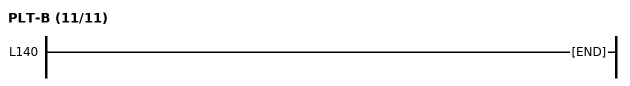
; L140
END

PROGRAM NG_CHUTE (task: 스캔 프로그램)

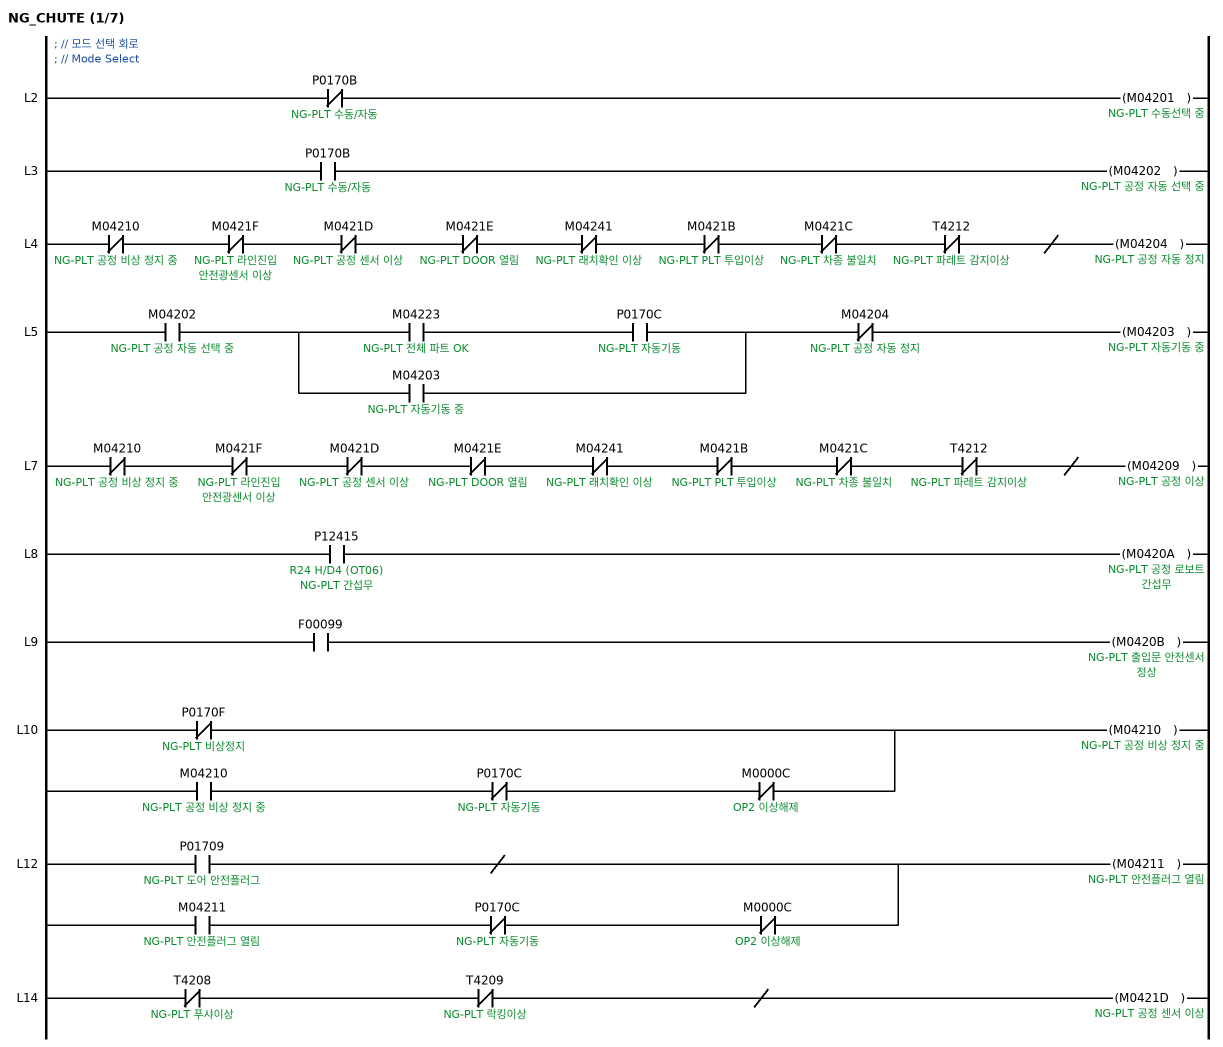
// // 모드 선택 회로
//   // Mode Select
; L2
LOAD NOT  P0170B	// NG-PLT 수동/자동
OUT       M04201	// NG-PLT 수동선택 중
; L3
LOAD      P0170B	// NG-PLT 수동/자동
OUT       M04202	// NG-PLT 공정 자동 선택 중
; L4
LOAD NOT  M04210	// NG-PLT 공정 비상 정지 중
AND NOT   M0421F	// NG-PLT 라인진입 안전광센서 이상
AND NOT   M0421D	// NG-PLT 공정 센서 이상
AND NOT   M0421E	// NG-PLT DOOR 열림
AND NOT   M04241	// NG-PLT 래치확인 이상
AND NOT   M0421B	// NG-PLT PLT 투입이상
AND NOT   M0421C	// NG-PLT 차종 불일치
AND NOT   T4212	// NG-PLT 파레트 감지이상
NOT
OUT       M04204	// NG-PLT 공정 자동 정지
; L5
LOAD      M04202	// NG-PLT 공정 자동 선택 중
LOAD      M04223	// NG-PLT 전체 파트 OK
AND       P0170C	// NG-PLT 자동기동
OR        M04203	// NG-PLT 자동기동 중
AND LOAD
AND NOT   M04204	// NG-PLT 공정 자동 정지
OUT       M04203	// NG-PLT 자동기동 중
; L7
LOAD NOT  M04210	// NG-PLT 공정 비상 정지 중
AND NOT   M0421F	// NG-PLT 라인진입 안전광센서 이상
AND NOT   M0421D	// NG-PLT 공정 센서 이상
AND NOT   M0421E	// NG-PLT DOOR 열림
AND NOT   M04241	// NG-PLT 래치확인 이상
AND NOT   M0421B	// NG-PLT PLT 투입이상
AND NOT   M0421C	// NG-PLT 차종 불일치
AND NOT   T4212	// NG-PLT 파레트 감지이상
NOT
OUT       M04209	// NG-PLT 공정 이상
; L8
LOAD      P12415	// R24 H/D4 (OT06) NG-PLT 간섭무
OUT       M0420A	// NG-PLT 공정 로보트 간섭무
; L9
LOAD      F00099
OUT       M0420B	// NG-PLT 출입문 안전센서 정상
; L10
LOAD NOT  P0170F	// NG-PLT 비상정지
LOAD      M04210	// NG-PLT 공정 비상 정지 중
AND NOT   P0170C	// NG-PLT 자동기동
AND NOT   M0000C	// OP2 이상해제
OR LOAD
OUT       M04210	// NG-PLT 공정 비상 정지 중
; L12
LOAD      P01709	// NG-PLT 도어 안전플러그
NOT
LOAD      M04211	// NG-PLT 안전플러그 열림
AND NOT   P0170C	// NG-PLT 자동기동
AND NOT   M0000C	// OP2 이상해제
OR LOAD
OUT       M04211	// NG-PLT 안전플러그 열림
; L14
LOAD NOT  T4208	// NG-PLT 푸샤이상
AND NOT   T4209	// NG-PLT 락킹이상
NOT
OUT       M0421D	// NG-PLT 공정 센서 이상

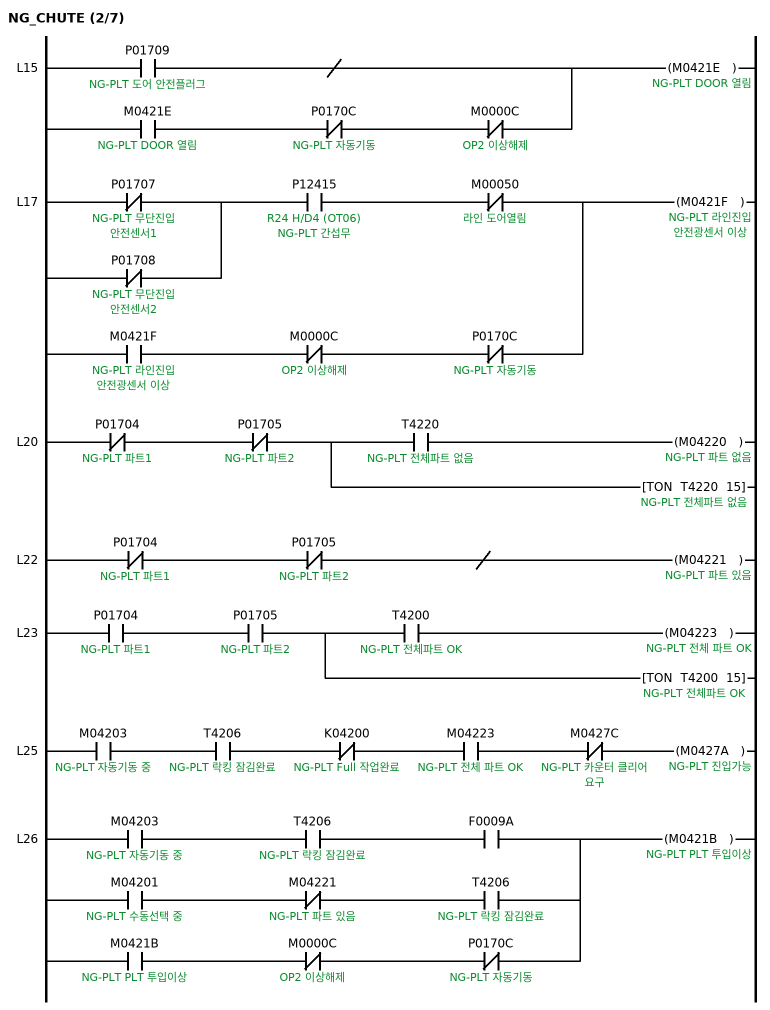
; L15
LOAD      P01709	// NG-PLT 도어 안전플러그
NOT
LOAD      M0421E	// NG-PLT DOOR 열림
AND NOT   P0170C	// NG-PLT 자동기동
AND NOT   M0000C	// OP2 이상해제
OR LOAD
OUT       M0421E	// NG-PLT DOOR 열림
; L17
LOAD NOT  P01707	// NG-PLT 무단진입 안전센서1
OR NOT    P01708	// NG-PLT 무단진입 안전센서2
AND       P12415	// R24 H/D4 (OT06) NG-PLT 간섭무
AND NOT   M00050	// 라인 도어열림
LOAD      M0421F	// NG-PLT 라인진입 안전광센서 이상
AND NOT   M0000C	// OP2 이상해제
AND NOT   P0170C	// NG-PLT 자동기동
OR LOAD
OUT       M0421F	// NG-PLT 라인진입 안전광센서 이상
; L20
LOAD NOT  P01704	// NG-PLT 파트1
AND NOT   P01705	// NG-PLT 파트2
MPUSH
AND       T4220	// NG-PLT 전체파트 없음
OUT       M04220	// NG-PLT 파트 없음
MPOP
TON       T4220 15	// NG-PLT 전체파트 없음
; L22
LOAD NOT  P01704	// NG-PLT 파트1
AND NOT   P01705	// NG-PLT 파트2
NOT
OUT       M04221	// NG-PLT 파트 있음
; L23
LOAD      P01704	// NG-PLT 파트1
AND       P01705	// NG-PLT 파트2
MPUSH
AND       T4200	// NG-PLT 전체파트 OK
OUT       M04223	// NG-PLT 전체 파트 OK
MPOP
TON       T4200 15	// NG-PLT 전체파트 OK
; L25
LOAD      M04203	// NG-PLT 자동기동 중
AND       T4206	// NG-PLT 락킹 잠김완료
AND NOT   K04200	// NG-PLT Full 작업완료
AND       M04223	// NG-PLT 전체 파트 OK
AND NOT   M0427C	// NG-PLT 카운터 클리어 요구
OUT       M0427A	// NG-PLT 진입가능
; L26
LOAD      M04203	// NG-PLT 자동기동 중
AND       T4206	// NG-PLT 락킹 잠김완료
AND       F0009A
LOAD      M04201	// NG-PLT 수동선택 중
AND NOT   M04221	// NG-PLT 파트 있음
AND       T4206	// NG-PLT 락킹 잠김완료
OR LOAD
LOAD      M0421B	// NG-PLT PLT 투입이상
AND NOT   M0000C	// OP2 이상해제
AND NOT   P0170C	// NG-PLT 자동기동
OR LOAD
OUT       M0421B	// NG-PLT PLT 투입이상

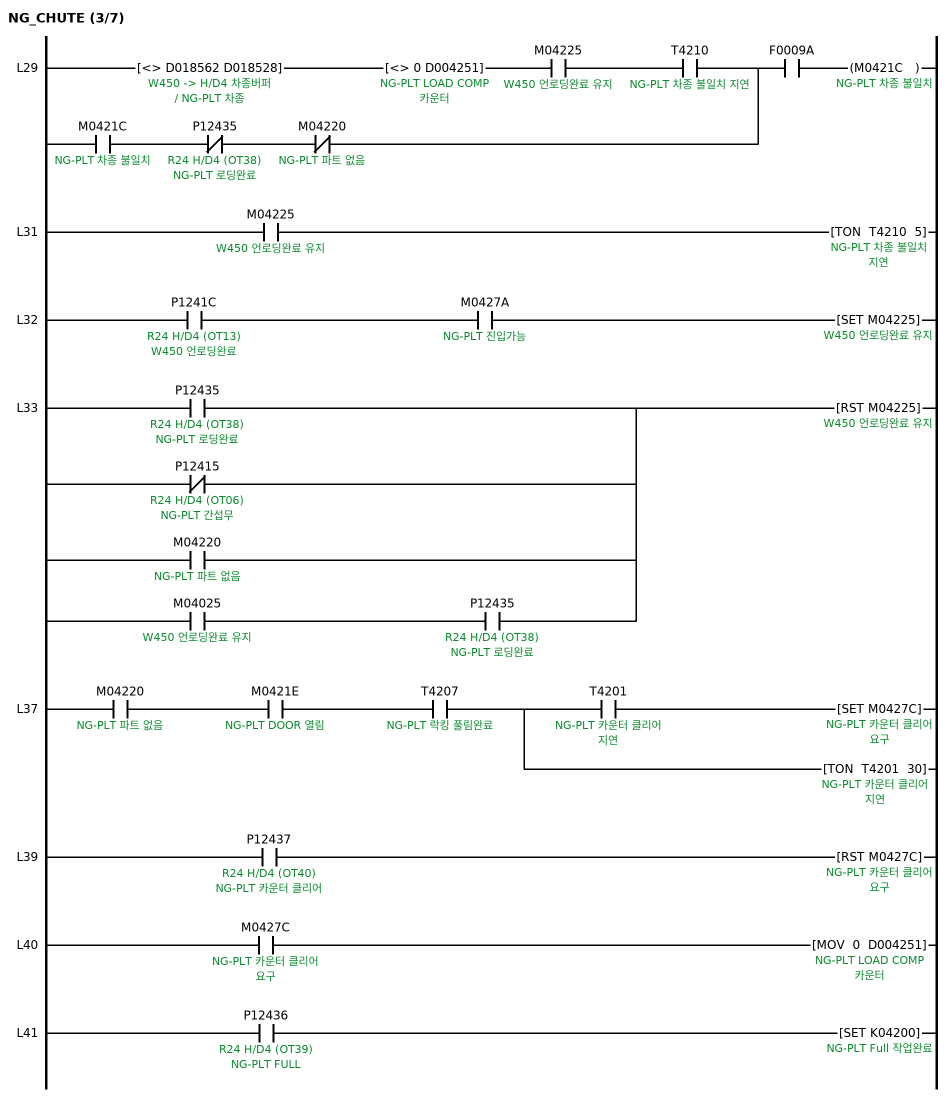
; L29
LOAD<>    D018562 D018528	// W450 -> H/D4 차종버퍼 / NG-PLT 차종
AND<>     0 D004251	// NG-PLT LOAD COMP 카운터
AND       M04225	// W450 언로딩완료 유지
AND       T4210	// NG-PLT 차종 불일치 지연
LOAD      M0421C	// NG-PLT 차종 불일치
AND NOT   P12435	// R24 H/D4 (OT38) NG-PLT 로딩완료
AND NOT   M04220	// NG-PLT 파트 없음
OR LOAD
AND       F0009A
OUT       M0421C	// NG-PLT 차종 불일치
; L31
LOAD      M04225	// W450 언로딩완료 유지
TON       T4210 5	// NG-PLT 차종 불일치 지연
; L32
LOAD      P1241C	// R24 H/D4 (OT13) W450 언로딩완료
AND       M0427A	// NG-PLT 진입가능
SET       M04225	// W450 언로딩완료 유지
; L33
LOAD      P12435	// R24 H/D4 (OT38) NG-PLT 로딩완료
OR NOT    P12415	// R24 H/D4 (OT06) NG-PLT 간섭무
OR        M04220	// NG-PLT 파트 없음
LOAD      M04025	// W450 언로딩완료 유지
AND       P12435	// R24 H/D4 (OT38) NG-PLT 로딩완료
OR LOAD
RST       M04225	// W450 언로딩완료 유지
; L37
LOAD      M04220	// NG-PLT 파트 없음
AND       M0421E	// NG-PLT DOOR 열림
AND       T4207	// NG-PLT 락킹 풀림완료
MPUSH
AND       T4201	// NG-PLT 카운터 클리어 지연
SET       M0427C	// NG-PLT 카운터 클리어 요구
MPOP
TON       T4201 30	// NG-PLT 카운터 클리어 지연
; L39
LOAD      P12437	// R24 H/D4 (OT40) NG-PLT 카운터 클리어
RST       M0427C	// NG-PLT 카운터 클리어 요구
; L40
LOAD      M0427C	// NG-PLT 카운터 클리어 요구
MOV       0 D004251	// NG-PLT LOAD COMP 카운터
; L41
LOAD      P12436	// R24 H/D4 (OT39) NG-PLT FULL
SET       K04200	// NG-PLT Full 작업완료

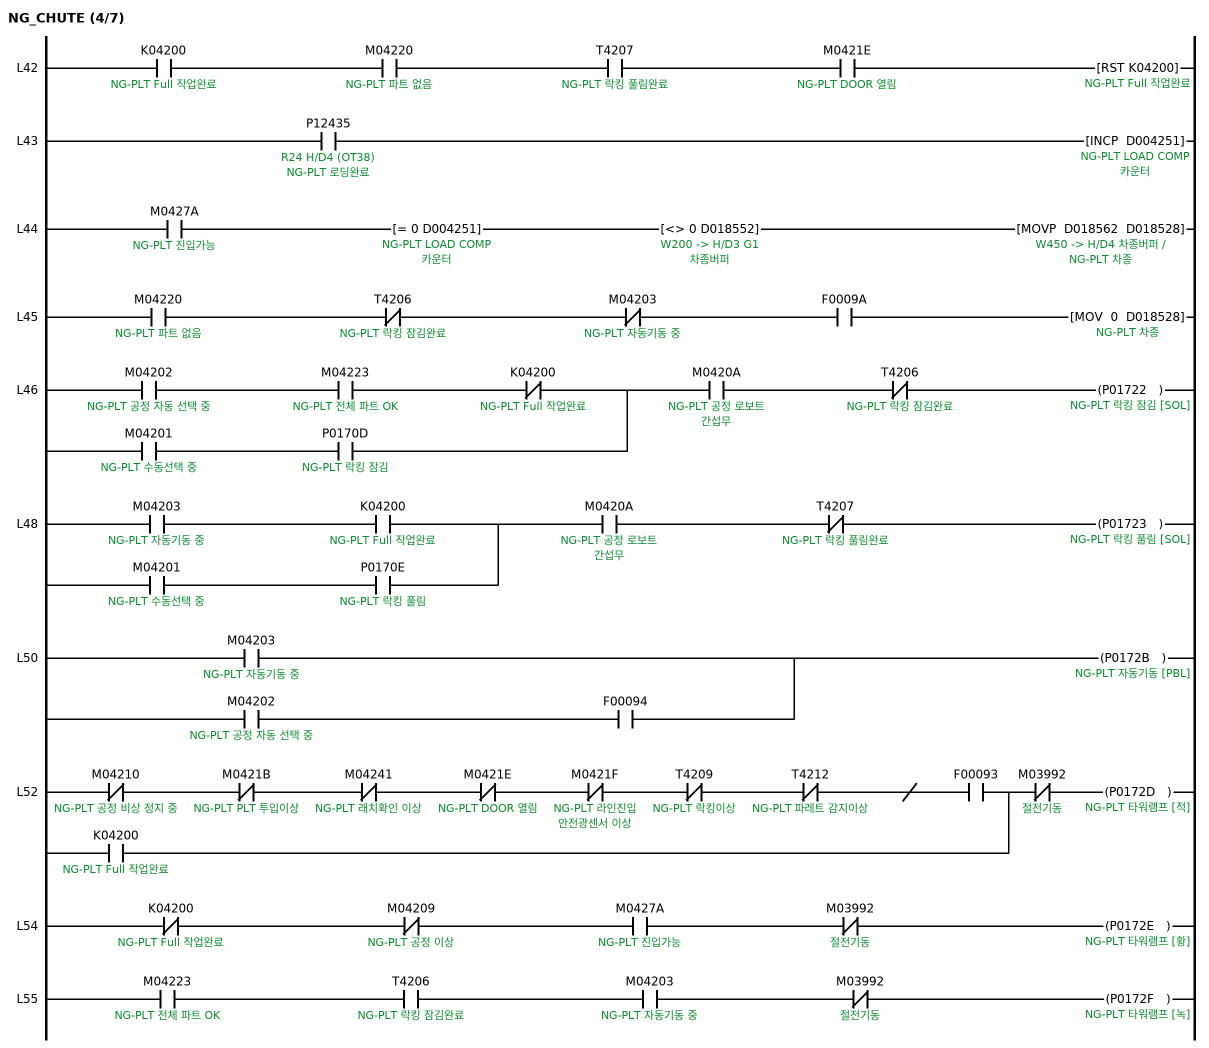
; L42
LOAD      K04200	// NG-PLT Full 작업완료
AND       M04220	// NG-PLT 파트 없음
AND       T4207	// NG-PLT 락킹 풀림완료
AND       M0421E	// NG-PLT DOOR 열림
RST       K04200	// NG-PLT Full 작업완료
; L43
LOAD      P12435	// R24 H/D4 (OT38) NG-PLT 로딩완료
INCP      D004251	// NG-PLT LOAD COMP 카운터
; L44
LOAD      M0427A	// NG-PLT 진입가능
AND=      0 D004251	// NG-PLT LOAD COMP 카운터
AND<>     0 D018552	// W200 -> H/D3 G1 차종버퍼
MOVP      D018562 D018528	// W450 -> H/D4 차종버퍼 / NG-PLT 차종
; L45
LOAD      M04220	// NG-PLT 파트 없음
AND NOT   T4206	// NG-PLT 락킹 잠김완료
AND NOT   M04203	// NG-PLT 자동기동 중
AND       F0009A
MOV       0 D018528	// NG-PLT 차종
; L46
LOAD      M04202	// NG-PLT 공정 자동 선택 중
AND       M04223	// NG-PLT 전체 파트 OK
AND NOT   K04200	// NG-PLT Full 작업완료
LOAD      M04201	// NG-PLT 수동선택 중
AND       P0170D	// NG-PLT 락킹 잠김
OR LOAD
AND       M0420A	// NG-PLT 공정 로보트 간섭무
AND NOT   T4206	// NG-PLT 락킹 잠김완료
OUT       P01722	// NG-PLT 락킹 잠김 [SOL]
; L48
LOAD      M04203	// NG-PLT 자동기동 중
AND       K04200	// NG-PLT Full 작업완료
LOAD      M04201	// NG-PLT 수동선택 중
AND       P0170E	// NG-PLT 락킹 풀림
OR LOAD
AND       M0420A	// NG-PLT 공정 로보트 간섭무
AND NOT   T4207	// NG-PLT 락킹 풀림완료
OUT       P01723	// NG-PLT 락킹 풀림 [SOL]
; L50
LOAD      M04203	// NG-PLT 자동기동 중
LOAD      M04202	// NG-PLT 공정 자동 선택 중
AND       F00094
OR LOAD
OUT       P0172B	// NG-PLT 자동기동 [PBL]
; L52
LOAD NOT  M04210	// NG-PLT 공정 비상 정지 중
AND NOT   M0421B	// NG-PLT PLT 투입이상
AND NOT   M04241	// NG-PLT 래치확인 이상
AND NOT   M0421E	// NG-PLT DOOR 열림
AND NOT   M0421F	// NG-PLT 라인진입 안전광센서 이상
AND NOT   T4209	// NG-PLT 락킹이상
AND NOT   T4212	// NG-PLT 파레트 감지이상
NOT
AND       F00093
OR        K04200	// NG-PLT Full 작업완료
AND NOT   M03992	// 절전기동
OUT       P0172D	// NG-PLT 타워램프 [적]
; L54
LOAD NOT  K04200	// NG-PLT Full 작업완료
AND NOT   M04209	// NG-PLT 공정 이상
AND       M0427A	// NG-PLT 진입가능
AND NOT   M03992	// 절전기동
OUT       P0172E	// NG-PLT 타워램프 [황]
; L55
LOAD      M04223	// NG-PLT 전체 파트 OK
AND       T4206	// NG-PLT 락킹 잠김완료
AND       M04203	// NG-PLT 자동기동 중
AND NOT   M03992	// 절전기동
OUT       P0172F	// NG-PLT 타워램프 [녹]

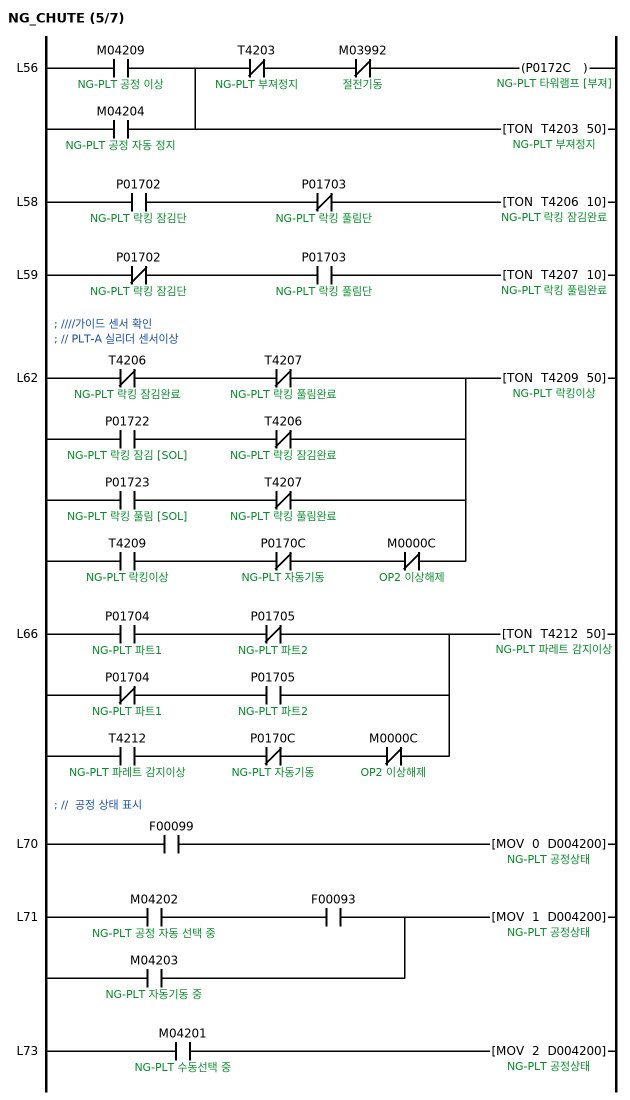
; L56
LOAD      M04209	// NG-PLT 공정 이상
OR        M04204	// NG-PLT 공정 자동 정지
MPUSH
AND NOT   T4203	// NG-PLT 부져정지
AND NOT   M03992	// 절전기동
OUT       P0172C	// NG-PLT 타워램프 [부져]
MPOP
TON       T4203 50	// NG-PLT 부져정지
; L58
LOAD      P01702	// NG-PLT 락킹 잠김단
AND NOT   P01703	// NG-PLT 락킹 풀림단
TON       T4206 10	// NG-PLT 락킹 잠김완료
; L59
LOAD NOT  P01702	// NG-PLT 락킹 잠김단
AND       P01703	// NG-PLT 락킹 풀림단
TON       T4207 10	// NG-PLT 락킹 풀림완료
// ////가이드 센서 확인
// // PLT-A 실리더 센서이상
; L62
LOAD NOT  T4206	// NG-PLT 락킹 잠김완료
AND NOT   T4207	// NG-PLT 락킹 풀림완료
LOAD      P01722	// NG-PLT 락킹 잠김 [SOL]
AND NOT   T4206	// NG-PLT 락킹 잠김완료
OR LOAD
LOAD      P01723	// NG-PLT 락킹 풀림 [SOL]
AND NOT   T4207	// NG-PLT 락킹 풀림완료
OR LOAD
LOAD      T4209	// NG-PLT 락킹이상
AND NOT   P0170C	// NG-PLT 자동기동
AND NOT   M0000C	// OP2 이상해제
OR LOAD
TON       T4209 50	// NG-PLT 락킹이상
; L66
LOAD      P01704	// NG-PLT 파트1
AND NOT   P01705	// NG-PLT 파트2
LOAD NOT  P01704	// NG-PLT 파트1
AND       P01705	// NG-PLT 파트2
OR LOAD
LOAD      T4212	// NG-PLT 파레트 감지이상
AND NOT   P0170C	// NG-PLT 자동기동
AND NOT   M0000C	// OP2 이상해제
OR LOAD
TON       T4212 50	// NG-PLT 파레트 감지이상
//   //  공정 상태 표시
; L70
LOAD      F00099
MOV       0 D004200	// NG-PLT 공정상태
; L71
LOAD      M04202	// NG-PLT 공정 자동 선택 중
AND       F00093
OR        M04203	// NG-PLT 자동기동 중
MOV       1 D004200	// NG-PLT 공정상태
; L73
LOAD      M04201	// NG-PLT 수동선택 중
MOV       2 D004200	// NG-PLT 공정상태

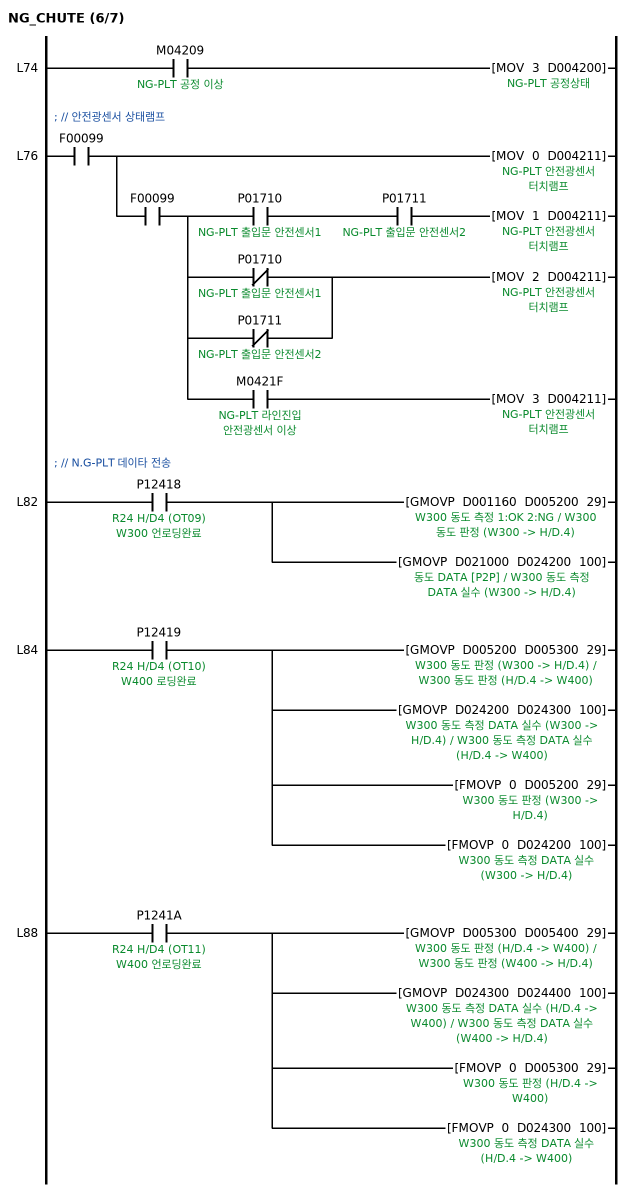
; L74
LOAD      M04209	// NG-PLT 공정 이상
MOV       3 D004200	// NG-PLT 공정상태
//   // 안전광센서 상태램프
; L76
LOAD      F00099
MOV       0 D004211	// NG-PLT 안전광센서 터치램프
AND       F00099
MPUSH
AND       P01710	// NG-PLT 출입문 안전센서1
AND       P01711	// NG-PLT 출입문 안전센서2
MOV       1 D004211	// NG-PLT 안전광센서 터치램프
MLOAD
LOAD NOT  P01710	// NG-PLT 출입문 안전센서1
OR NOT    P01711	// NG-PLT 출입문 안전센서2
AND LOAD
MOV       2 D004211	// NG-PLT 안전광센서 터치램프
MPOP
AND       M0421F	// NG-PLT 라인진입 안전광센서 이상
MOV       3 D004211	// NG-PLT 안전광센서 터치램프
//   // N.G-PLT 데이타 전송
; L82
LOAD      P12418	// R24 H/D4 (OT09) W300 언로딩완료
GMOVP     D001160 D005200 29	// W300 동도 측정 1:OK 2:NG / W300 동도 판정 (W300 -> H/D.4)
GMOVP     D021000 D024200 100	// 동도 DATA [P2P] / W300 동도 측정 DATA 실수 (W300 -> H/D.4)
; L84
LOAD      P12419	// R24 H/D4 (OT10) W400 로딩완료
GMOVP     D005200 D005300 29	// W300 동도 판정 (W300 -> H/D.4) / W300 동도 판정 (H/D.4 -> W400)
GMOVP     D024200 D024300 100	// W300 동도 측정 DATA 실수 (W300 -> H/D.4) / W300 동도 측정 DATA 실수 (H/D.4 -> W400)
FMOVP     0 D005200 29	// W300 동도 판정 (W300 -> H/D.4)
FMOVP     0 D024200 100	// W300 동도 측정 DATA 실수 (W300 -> H/D.4)
; L88
LOAD      P1241A	// R24 H/D4 (OT11) W400 언로딩완료
GMOVP     D005300 D005400 29	// W300 동도 판정 (H/D.4 -> W400) / W300 동도 판정 (W400 -> H/D.4)
GMOVP     D024300 D024400 100	// W300 동도 측정 DATA 실수 (H/D.4 -> W400) / W300 동도 측정 DATA 실수 (W400 -> H/D.4)
FMOVP     0 D005300 29	// W300 동도 판정 (H/D.4 -> W400)
FMOVP     0 D024300 100	// W300 동도 측정 DATA 실수 (H/D.4 -> W400)

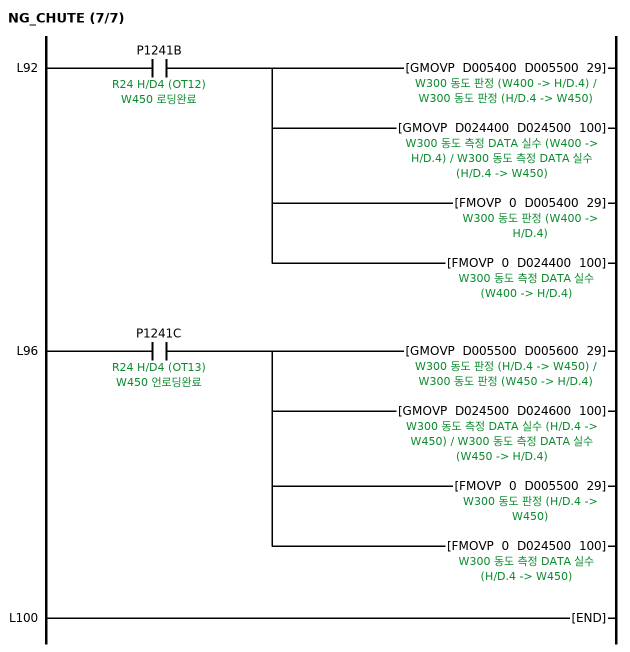
; L92
LOAD      P1241B	// R24 H/D4 (OT12) W450 로딩완료
GMOVP     D005400 D005500 29	// W300 동도 판정 (W400 -> H/D.4) / W300 동도 판정 (H/D.4 -> W450)
GMOVP     D024400 D024500 100	// W300 동도 측정 DATA 실수 (W400 -> H/D.4) / W300 동도 측정 DATA 실수 (H/D.4 -> W450)
FMOVP     0 D005400 29	// W300 동도 판정 (W400 -> H/D.4)
FMOVP     0 D024400 100	// W300 동도 측정 DATA 실수 (W400 -> H/D.4)
; L96
LOAD      P1241C	// R24 H/D4 (OT13) W450 언로딩완료
GMOVP     D005500 D005600 29	// W300 동도 판정 (H/D.4 -> W450) / W300 동도 판정 (W450 -> H/D.4)
GMOVP     D024500 D024600 100	// W300 동도 측정 DATA 실수 (H/D.4 -> W450) / W300 동도 측정 DATA 실수 (W450 -> H/D.4)
FMOVP     0 D005500 29	// W300 동도 판정 (H/D.4 -> W450)
FMOVP     0 D024500 100	// W300 동도 측정 DATA 실수 (H/D.4 -> W450)
; L100
END

PROGRAM OK_NG_Master (task: 스캔 프로그램)

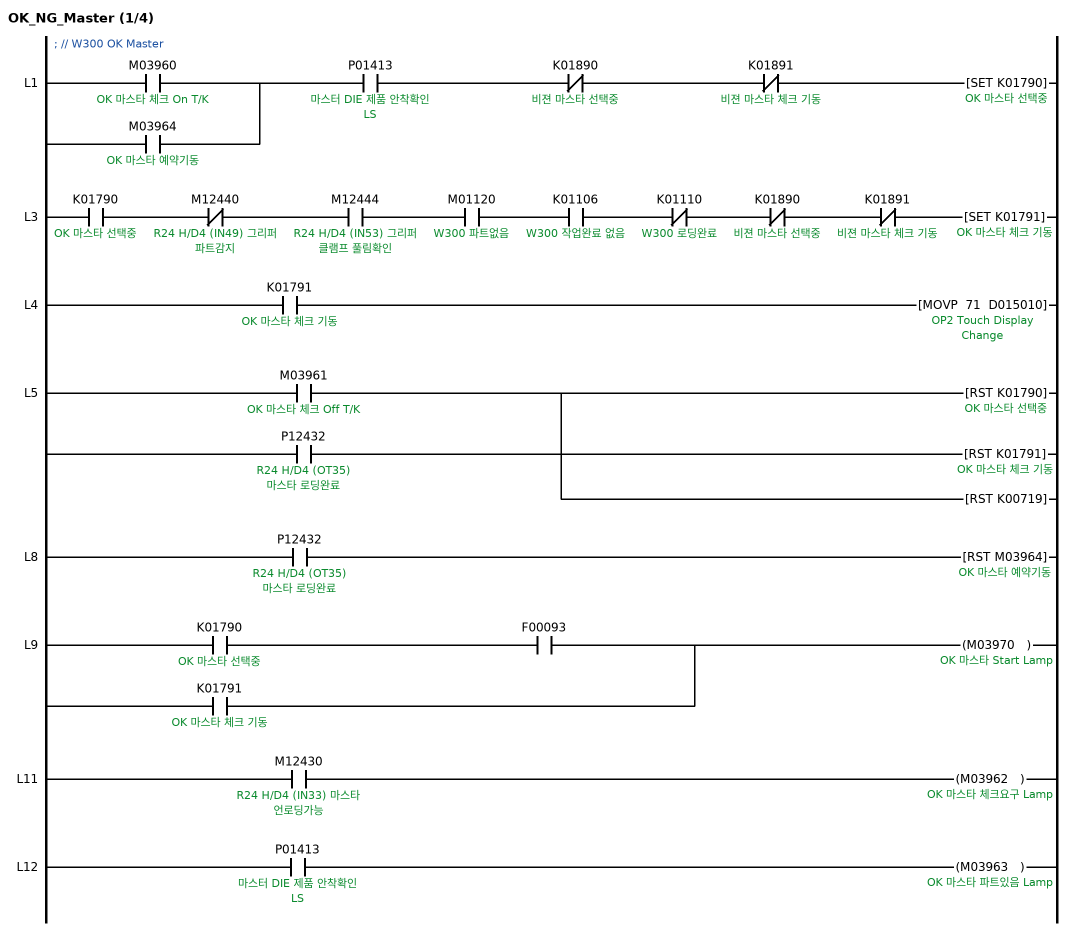
//   // W300 OK Master
; L1
LOAD      M03960	// OK 마스타 체크 On T/K
OR        M03964	// OK 마스타 예약기동
AND       P01413	// 마스터 DIE 제품 안착확인 LS
AND NOT   K01890	// 비젼 마스타 선택중
AND NOT   K01891	// 비젼 마스타 체크 기동
SET       K01790	// OK 마스타 선택중
; L3
LOAD      K01790	// OK 마스타 선택중
AND NOT   M12440	// R24 H/D4 (IN49) 그리퍼 파트감지
AND       M12444	// R24 H/D4 (IN53) 그리퍼 클램프 풀림확인
AND       M01120	// W300 파트없음
AND       K01106	// W300 작업완료 없음
AND NOT   K01110	// W300 로딩완료
AND NOT   K01890	// 비젼 마스타 선택중
AND NOT   K01891	// 비젼 마스타 체크 기동
SET       K01791	// OK 마스타 체크 기동
; L4
LOAD      K01791	// OK 마스타 체크 기동
MOVP      71 D015010	// OP2 Touch Display Change
; L5
LOAD      M03961	// OK 마스타 체크 Off T/K
OR        P12432	// R24 H/D4 (OT35) 마스타 로딩완료
RST       K01790	// OK 마스타 선택중
RST       K01791	// OK 마스타 체크 기동
RST       K00719
; L8
LOAD      P12432	// R24 H/D4 (OT35) 마스타 로딩완료
RST       M03964	// OK 마스타 예약기동
; L9
LOAD      K01790	// OK 마스타 선택중
AND       F00093
OR        K01791	// OK 마스타 체크 기동
OUT       M03970	// OK 마스타 Start Lamp
; L11
LOAD      M12430	// R24 H/D4 (IN33) 마스타 언로딩가능
OUT       M03962	// OK 마스타 체크요구 Lamp
; L12
LOAD      P01413	// 마스터 DIE 제품 안착확인 LS
OUT       M03963	// OK 마스타 파트있음 Lamp

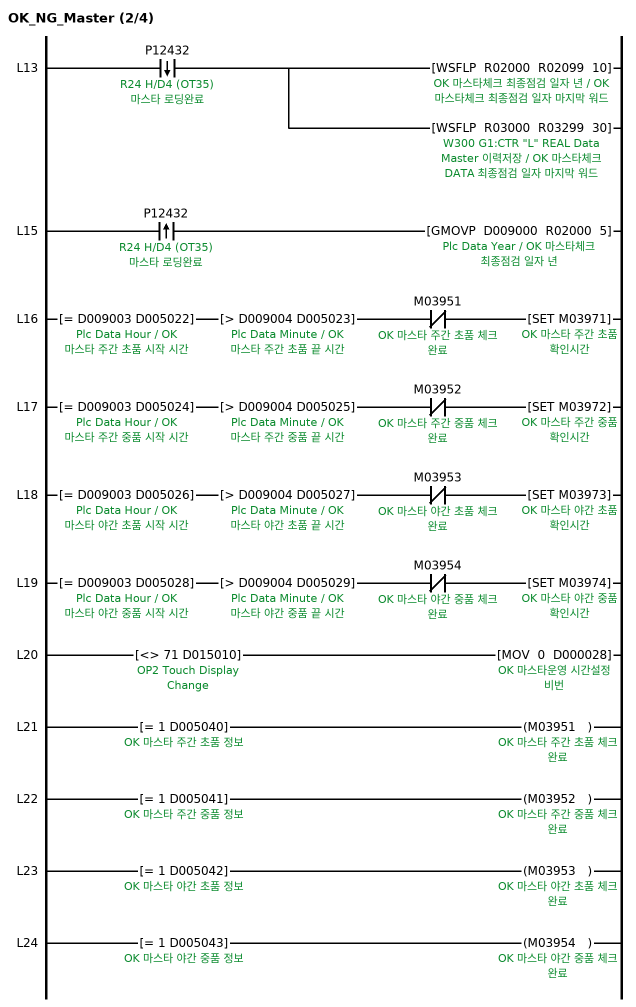
; L13
LOADN     P12432	// R24 H/D4 (OT35) 마스타 로딩완료
WSFLP     R02000 R02099 10	// OK 마스타체크 최종점검 일자 년 / OK 마스타체크 최종점검 일자 마지막 워드
WSFLP     R03000 R03299 30	// W300 G1:CTR "L" REAL Data Master 이력저장 / OK 마스타체크 DATA 최종점검 일자 마지막 워드
; L15
LOADP     P12432	// R24 H/D4 (OT35) 마스타 로딩완료
GMOVP     D009000 R02000 5	// Plc Data Year / OK 마스타체크 최종점검 일자 년
; L16
LOAD=     D009003 D005022	// Plc Data Hour / OK 마스타 주간 초품 시작 시간
AND>      D009004 D005023	// Plc Data Minute / OK 마스타 주간 초품 끝 시간
AND NOT   M03951	// OK 마스타 주간 초품 체크 완료
SET       M03971	// OK 마스타 주간 초품 확인시간
; L17
LOAD=     D009003 D005024	// Plc Data Hour / OK 마스타 주간 중품 시작 시간
AND>      D009004 D005025	// Plc Data Minute / OK 마스타 주간 중품 끝 시간
AND NOT   M03952	// OK 마스타 주간 중품 체크 완료
SET       M03972	// OK 마스타 주간 중품 확인시간
; L18
LOAD=     D009003 D005026	// Plc Data Hour / OK 마스타 야간 초품 시작 시간
AND>      D009004 D005027	// Plc Data Minute / OK 마스타 야간 초품 끝 시간
AND NOT   M03953	// OK 마스타 야간 초품 체크 완료
SET       M03973	// OK 마스타 야간 초품 확인시간
; L19
LOAD=     D009003 D005028	// Plc Data Hour / OK 마스타 야간 중품 시작 시간
AND>      D009004 D005029	// Plc Data Minute / OK 마스타 야간 중품 끝 시간
AND NOT   M03954	// OK 마스타 야간 중품 체크 완료
SET       M03974	// OK 마스타 야간 중품 확인시간
; L20
LOAD<>    71 D015010	// OP2 Touch Display Change
MOV       0 D000028	// OK 마스타운영 시간설정 비번
; L21
LOAD=     1 D005040	// OK 마스타 주간 초품 정보
OUT       M03951	// OK 마스타 주간 초품 체크 완료
; L22
LOAD=     1 D005041	// OK 마스타 주간 중품 정보
OUT       M03952	// OK 마스타 주간 중품 체크 완료
; L23
LOAD=     1 D005042	// OK 마스타 야간 초품 정보
OUT       M03953	// OK 마스타 야간 초품 체크 완료
; L24
LOAD=     1 D005043	// OK 마스타 야간 중품 정보
OUT       M03954	// OK 마스타 야간 중품 체크 완료

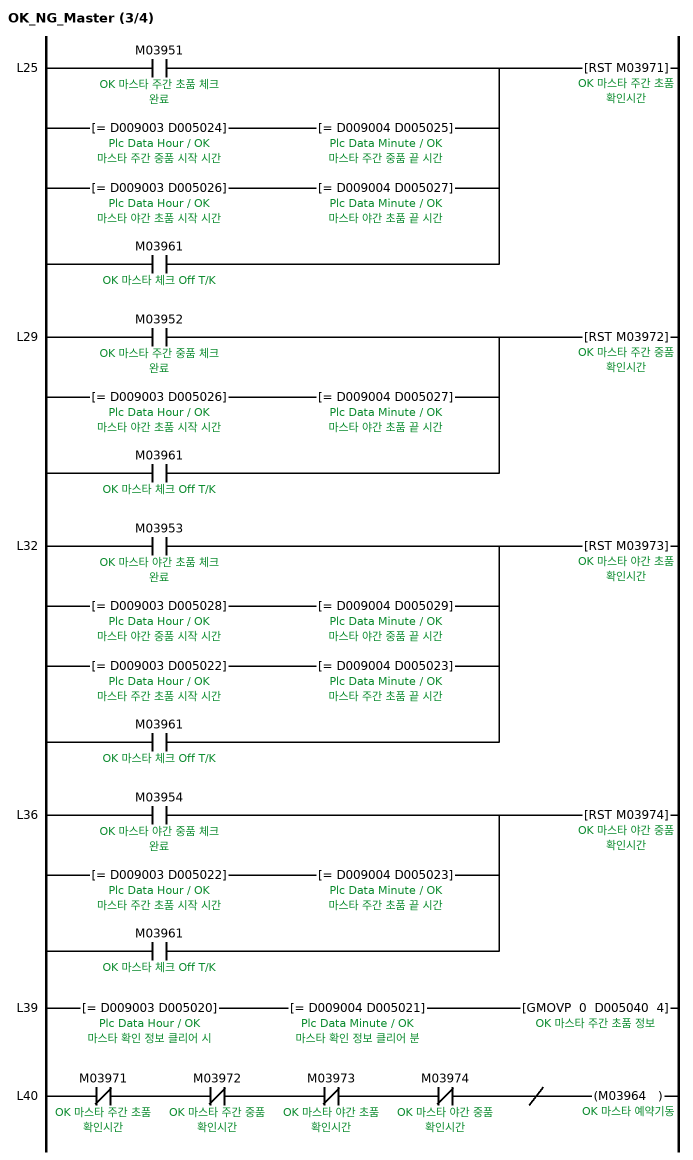
; L25
LOAD      M03951	// OK 마스타 주간 초품 체크 완료
LOAD=     D009003 D005024	// Plc Data Hour / OK 마스타 주간 중품 시작 시간
AND=      D009004 D005025	// Plc Data Minute / OK 마스타 주간 중품 끝 시간
OR LOAD
LOAD=     D009003 D005026	// Plc Data Hour / OK 마스타 야간 초품 시작 시간
AND=      D009004 D005027	// Plc Data Minute / OK 마스타 야간 초품 끝 시간
OR LOAD
OR        M03961	// OK 마스타 체크 Off T/K
RST       M03971	// OK 마스타 주간 초품 확인시간
; L29
LOAD      M03952	// OK 마스타 주간 중품 체크 완료
LOAD=     D009003 D005026	// Plc Data Hour / OK 마스타 야간 초품 시작 시간
AND=      D009004 D005027	// Plc Data Minute / OK 마스타 야간 초품 끝 시간
OR LOAD
OR        M03961	// OK 마스타 체크 Off T/K
RST       M03972	// OK 마스타 주간 중품 확인시간
; L32
LOAD      M03953	// OK 마스타 야간 초품 체크 완료
LOAD=     D009003 D005028	// Plc Data Hour / OK 마스타 야간 중품 시작 시간
AND=      D009004 D005029	// Plc Data Minute / OK 마스타 야간 중품 끝 시간
OR LOAD
LOAD=     D009003 D005022	// Plc Data Hour / OK 마스타 주간 초품 시작 시간
AND=      D009004 D005023	// Plc Data Minute / OK 마스타 주간 초품 끝 시간
OR LOAD
OR        M03961	// OK 마스타 체크 Off T/K
RST       M03973	// OK 마스타 야간 초품 확인시간
; L36
LOAD      M03954	// OK 마스타 야간 중품 체크 완료
LOAD=     D009003 D005022	// Plc Data Hour / OK 마스타 주간 초품 시작 시간
AND=      D009004 D005023	// Plc Data Minute / OK 마스타 주간 초품 끝 시간
OR LOAD
OR        M03961	// OK 마스타 체크 Off T/K
RST       M03974	// OK 마스타 야간 중품 확인시간
; L39
LOAD=     D009003 D005020	// Plc Data Hour / OK 마스타 확인 정보 클리어 시
AND=      D009004 D005021	// Plc Data Minute / OK 마스타 확인 정보 클리어 분
GMOVP     0 D005040 4	// OK 마스타 주간 초품 정보
; L40
LOAD NOT  M03971	// OK 마스타 주간 초품 확인시간
AND NOT   M03972	// OK 마스타 주간 중품 확인시간
AND NOT   M03973	// OK 마스타 야간 초품 확인시간
AND NOT   M03974	// OK 마스타 야간 중품 확인시간
NOT
OUT       M03964	// OK 마스타 예약기동

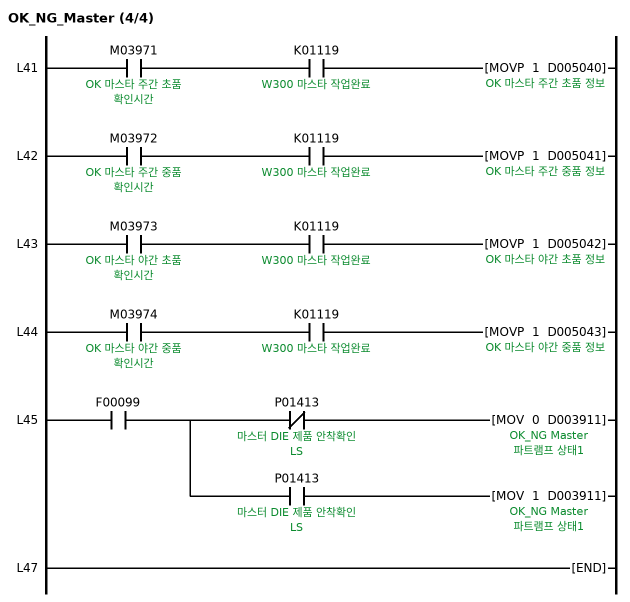
; L41
LOAD      M03971	// OK 마스타 주간 초품 확인시간
AND       K01119	// W300 마스타 작업완료
MOVP      1 D005040	// OK 마스타 주간 초품 정보
; L42
LOAD      M03972	// OK 마스타 주간 중품 확인시간
AND       K01119	// W300 마스타 작업완료
MOVP      1 D005041	// OK 마스타 주간 중품 정보
; L43
LOAD      M03973	// OK 마스타 야간 초품 확인시간
AND       K01119	// W300 마스타 작업완료
MOVP      1 D005042	// OK 마스타 야간 초품 정보
; L44
LOAD      M03974	// OK 마스타 야간 중품 확인시간
AND       K01119	// W300 마스타 작업완료
MOVP      1 D005043	// OK 마스타 야간 중품 정보
; L45
LOAD      F00099
MPUSH
AND NOT   P01413	// 마스터 DIE 제품 안착확인 LS
MOV       0 D003911	// OK_NG Master 파트램프 상태1
MPOP
AND       P01413	// 마스터 DIE 제품 안착확인 LS
MOV       1 D003911	// OK_NG Master 파트램프 상태1
; L47
END

PROGRAM SERVO_1_W100 (task: 스캔 프로그램)

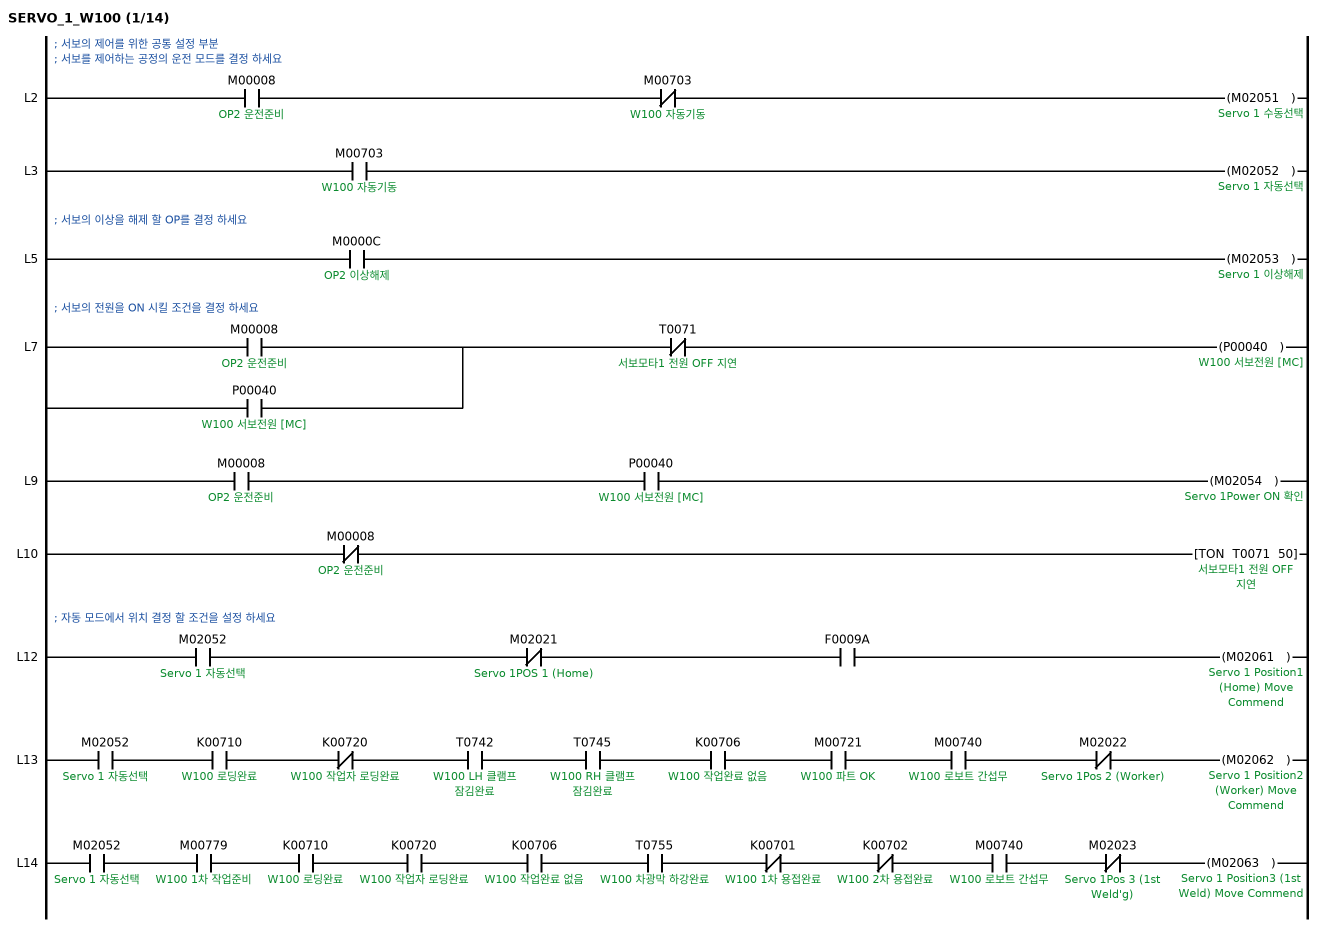
// 서보의 제어를 위한 공통 설정 부분
//     서보를 제어하는 공정의 운전 모드를 결정 하세요
; L2
LOAD      M00008	// OP2 운전준비
AND NOT   M00703	// W100 자동기동
OUT       M02051	// Servo 1 수동선택
; L3
LOAD      M00703	// W100 자동기동
OUT       M02052	// Servo 1 자동선택
//     서보의 이상을 해제 할 OP를 결정 하세요
; L5
LOAD      M0000C	// OP2 이상해제
OUT       M02053	// Servo 1 이상해제
//     서보의 전원을 ON 시킬 조건을 결정 하세요
; L7
LOAD      M00008	// OP2 운전준비
OR        P00040	// W100 서보전원 [MC]
AND NOT   T0071	// 서보모타1 전원 OFF 지연
OUT       P00040	// W100 서보전원 [MC]
; L9
LOAD      M00008	// OP2 운전준비
AND       P00040	// W100 서보전원 [MC]
OUT       M02054	// Servo 1Power ON 확인
; L10
LOAD NOT  M00008	// OP2 운전준비
TON       T0071 50	// 서보모타1 전원 OFF 지연
//     자동 모드에서 위치 결정 할 조건을 설정 하세요
; L12
LOAD      M02052	// Servo 1 자동선택
AND NOT   M02021	// Servo 1POS 1 (Home)
AND       F0009A
OUT       M02061	// Servo 1 Position1 (Home) Move Commend
; L13
LOAD      M02052	// Servo 1 자동선택
AND       K00710	// W100 로딩완료
AND NOT   K00720	// W100 작업자 로딩완료
AND       T0742	// W100 LH 클램프 잠김완료
AND       T0745	// W100 RH 클램프 잠김완료
AND       K00706	// W100 작업완료 없음
AND       M00721	// W100 파트 OK
AND       M00740	// W100 로보트 간섭무
AND NOT   M02022	// Servo 1Pos 2 (Worker)
OUT       M02062	// Servo 1 Position2 (Worker) Move Commend
; L14
LOAD      M02052	// Servo 1 자동선택
AND       M00779	// W100 1차 작업준비
AND       K00710	// W100 로딩완료
AND       K00720	// W100 작업자 로딩완료
AND       K00706	// W100 작업완료 없음
AND       T0755	// W100 차광막 하강완료
AND NOT   K00701	// W100 1차 용접완료
AND NOT   K00702	// W100 2차 용접완료
AND       M00740	// W100 로보트 간섭무
AND NOT   M02023	// Servo 1Pos 3 (1st Weld'g)
OUT       M02063	// Servo 1 Position3 (1st Weld) Move Commend

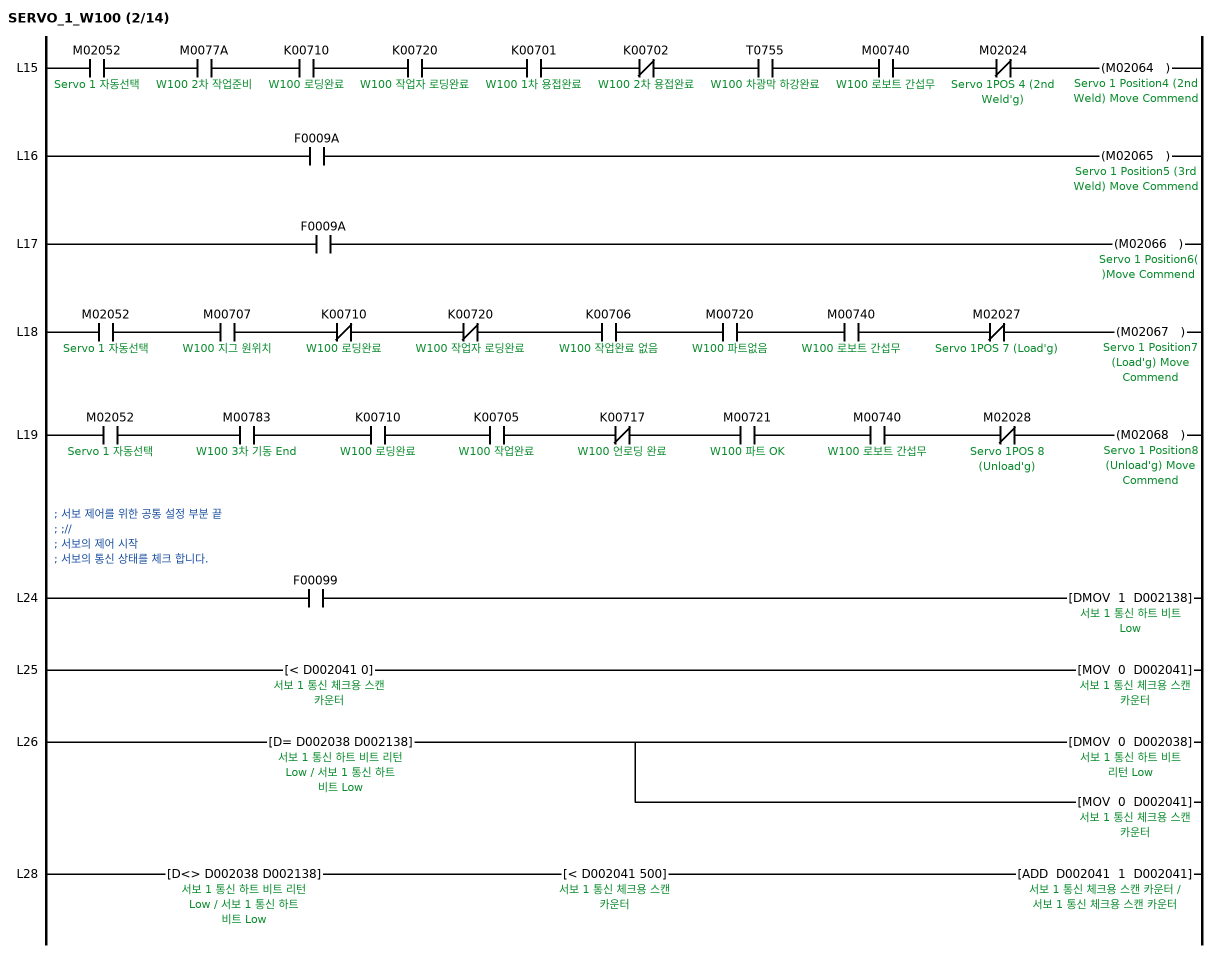
; L15
LOAD      M02052	// Servo 1 자동선택
AND       M0077A	// W100 2차 작업준비
AND       K00710	// W100 로딩완료
AND       K00720	// W100 작업자 로딩완료
AND       K00701	// W100 1차 용접완료
AND NOT   K00702	// W100 2차 용접완료
AND       T0755	// W100 차광막 하강완료
AND       M00740	// W100 로보트 간섭무
AND NOT   M02024	// Servo 1POS 4 (2nd Weld'g)
OUT       M02064	// Servo 1 Position4 (2nd Weld) Move Commend
; L16
LOAD      F0009A
OUT       M02065	// Servo 1 Position5 (3rd Weld) Move Commend
; L17
LOAD      F0009A
OUT       M02066	// Servo 1 Position6()Move Commend
; L18
LOAD      M02052	// Servo 1 자동선택
AND       M00707	// W100 지그 원위치
AND NOT   K00710	// W100 로딩완료
AND NOT   K00720	// W100 작업자 로딩완료
AND       K00706	// W100 작업완료 없음
AND       M00720	// W100 파트없음
AND       M00740	// W100 로보트 간섭무
AND NOT   M02027	// Servo 1POS 7 (Load'g)
OUT       M02067	// Servo 1 Position7 (Load'g) Move Commend
; L19
LOAD      M02052	// Servo 1 자동선택
AND       M00783	// W100 3차 기동 End
AND       K00710	// W100 로딩완료
AND       K00705	// W100 작업완료
AND NOT   K00717	// W100 언로딩 완료
AND       M00721	// W100 파트 OK
AND       M00740	// W100 로보트 간섭무
AND NOT   M02028	// Servo 1POS 8 (Unload'g)
OUT       M02068	// Servo 1 Position8 (Unload'g) Move Commend
// 서보 제어를 위한 공통 설정 부분 끝
// ;//
// 서보의 제어 시작
//     서보의 통신 상태를 체크 합니다.
; L24
LOAD      F00099
DMOV      1 D002138	// 서보 1 통신 하트 비트 Low
; L25
LOAD<     D002041 0	// 서보 1 통신 체크용 스캔 카운터
MOV       0 D002041	// 서보 1 통신 체크용 스캔 카운터
; L26
LOADD=    D002038 D002138	// 서보 1 통신 하트 비트 리턴 Low / 서보 1 통신 하트 비트 Low
DMOV      0 D002038	// 서보 1 통신 하트 비트 리턴 Low
MOV       0 D002041	// 서보 1 통신 체크용 스캔 카운터
; L28
LOADD<>   D002038 D002138	// 서보 1 통신 하트 비트 리턴 Low / 서보 1 통신 하트 비트 Low
AND<      D002041 500	// 서보 1 통신 체크용 스캔 카운터
ADD       D002041 1 D002041	// 서보 1 통신 체크용 스캔 카운터 / 서보 1 통신 체크용 스캔 카운터

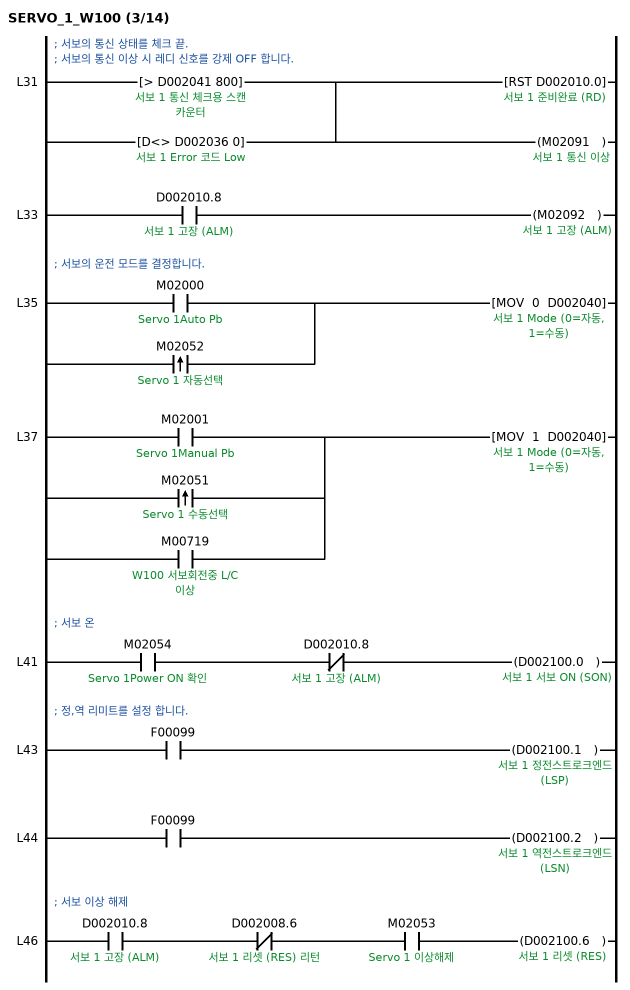
//     서보의 통신 상태를 체크 끝.
//     서보의 통신 이상 시 레디 신호를 강제 OFF 합니다.
; L31
LOAD>     D002041 800	// 서보 1 통신 체크용 스캔 카운터
ORD<>     D002036 0	// 서보 1 Error 코드 Low
RST       D002010.0	// 서보 1 준비완료 (RD)
OUT       M02091	// 서보 1 통신 이상
; L33
LOAD      D002010.8	// 서보 1 고장 (ALM)
OUT       M02092	// 서보 1 고장 (ALM)
//     서보의 운전 모드를 결정합니다.
; L35
LOAD      M02000	// Servo 1Auto Pb
ORP       M02052	// Servo 1 자동선택
MOV       0 D002040	// 서보 1 Mode (0=자동, 1=수동)
; L37
LOAD      M02001	// Servo 1Manual Pb
ORP       M02051	// Servo 1 수동선택
OR        M00719	// W100 서보회전중 L/C 이상
MOV       1 D002040	// 서보 1 Mode (0=자동, 1=수동)
//     서보 온
; L41
LOAD      M02054	// Servo 1Power ON 확인
AND NOT   D002010.8	// 서보 1 고장 (ALM)
OUT       D002100.0	// 서보 1 서보 ON (SON)
//     정,역 리미트를 설정 합니다.
; L43
LOAD      F00099
OUT       D002100.1	// 서보 1 정전스트로크엔드 (LSP)
; L44
LOAD      F00099
OUT       D002100.2	// 서보 1 역전스트로크엔드 (LSN)
//     서보 이상 해제
; L46
LOAD      D002010.8	// 서보 1 고장 (ALM)
AND NOT   D002008.6	// 서보 1 리셋 (RES) 리턴
AND       M02053	// Servo 1 이상해제
OUT       D002100.6	// 서보 1 리셋 (RES)

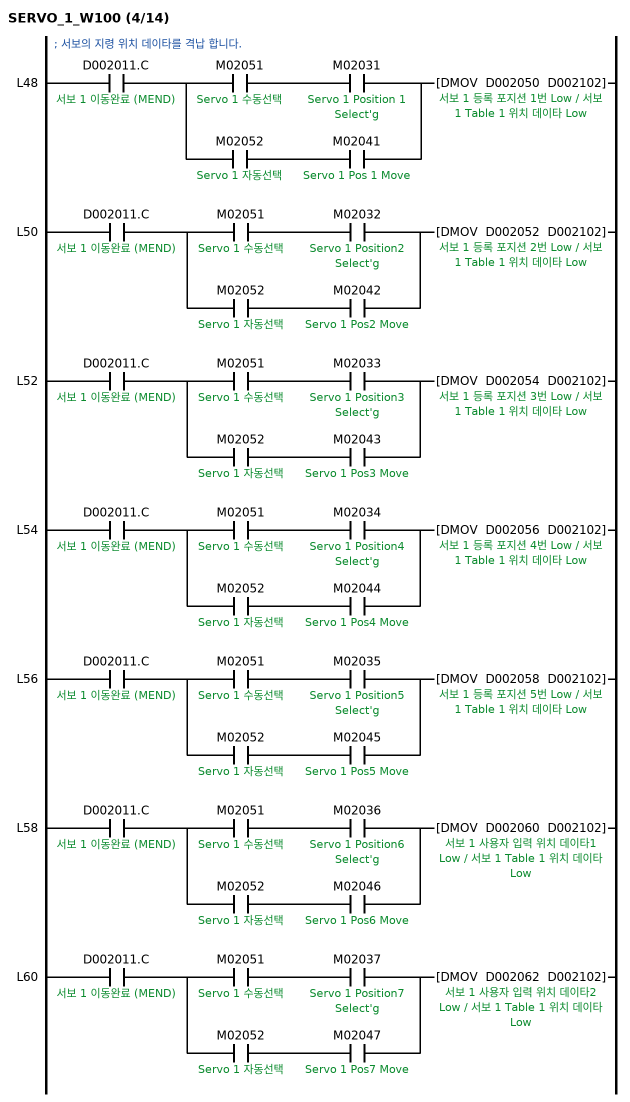
//     서보의 지령 위치 데이타를 격납 합니다.
; L48
LOAD      D002011.C	// 서보 1 이동완료 (MEND)
LOAD      M02051	// Servo 1 수동선택
AND       M02031	// Servo 1 Position 1 Select'g
LOAD      M02052	// Servo 1 자동선택
AND       M02041	// Servo 1 Pos 1 Move
OR LOAD
AND LOAD
DMOV      D002050 D002102	// 서보 1 등록 포지션 1번 Low / 서보 1 Table 1 위치 데이타 Low
; L50
LOAD      D002011.C	// 서보 1 이동완료 (MEND)
LOAD      M02051	// Servo 1 수동선택
AND       M02032	// Servo 1 Position2 Select'g
LOAD      M02052	// Servo 1 자동선택
AND       M02042	// Servo 1 Pos2 Move
OR LOAD
AND LOAD
DMOV      D002052 D002102	// 서보 1 등록 포지션 2번 Low / 서보 1 Table 1 위치 데이타 Low
; L52
LOAD      D002011.C	// 서보 1 이동완료 (MEND)
LOAD      M02051	// Servo 1 수동선택
AND       M02033	// Servo 1 Position3 Select'g
LOAD      M02052	// Servo 1 자동선택
AND       M02043	// Servo 1 Pos3 Move
OR LOAD
AND LOAD
DMOV      D002054 D002102	// 서보 1 등록 포지션 3번 Low / 서보 1 Table 1 위치 데이타 Low
; L54
LOAD      D002011.C	// 서보 1 이동완료 (MEND)
LOAD      M02051	// Servo 1 수동선택
AND       M02034	// Servo 1 Position4 Select'g
LOAD      M02052	// Servo 1 자동선택
AND       M02044	// Servo 1 Pos4 Move
OR LOAD
AND LOAD
DMOV      D002056 D002102	// 서보 1 등록 포지션 4번 Low / 서보 1 Table 1 위치 데이타 Low
; L56
LOAD      D002011.C	// 서보 1 이동완료 (MEND)
LOAD      M02051	// Servo 1 수동선택
AND       M02035	// Servo 1 Position5 Select'g
LOAD      M02052	// Servo 1 자동선택
AND       M02045	// Servo 1 Pos5 Move
OR LOAD
AND LOAD
DMOV      D002058 D002102	// 서보 1 등록 포지션 5번 Low / 서보 1 Table 1 위치 데이타 Low
; L58
LOAD      D002011.C	// 서보 1 이동완료 (MEND)
LOAD      M02051	// Servo 1 수동선택
AND       M02036	// Servo 1 Position6 Select'g
LOAD      M02052	// Servo 1 자동선택
AND       M02046	// Servo 1 Pos6 Move
OR LOAD
AND LOAD
DMOV      D002060 D002102	// 서보 1 사용자 입력 위치 데이타1 Low / 서보 1 Table 1 위치 데이타 Low
; L60
LOAD      D002011.C	// 서보 1 이동완료 (MEND)
LOAD      M02051	// Servo 1 수동선택
AND       M02037	// Servo 1 Position7 Select'g
LOAD      M02052	// Servo 1 자동선택
AND       M02047	// Servo 1 Pos7 Move
OR LOAD
AND LOAD
DMOV      D002062 D002102	// 서보 1 사용자 입력 위치 데이타2 Low / 서보 1 Table 1 위치 데이타 Low

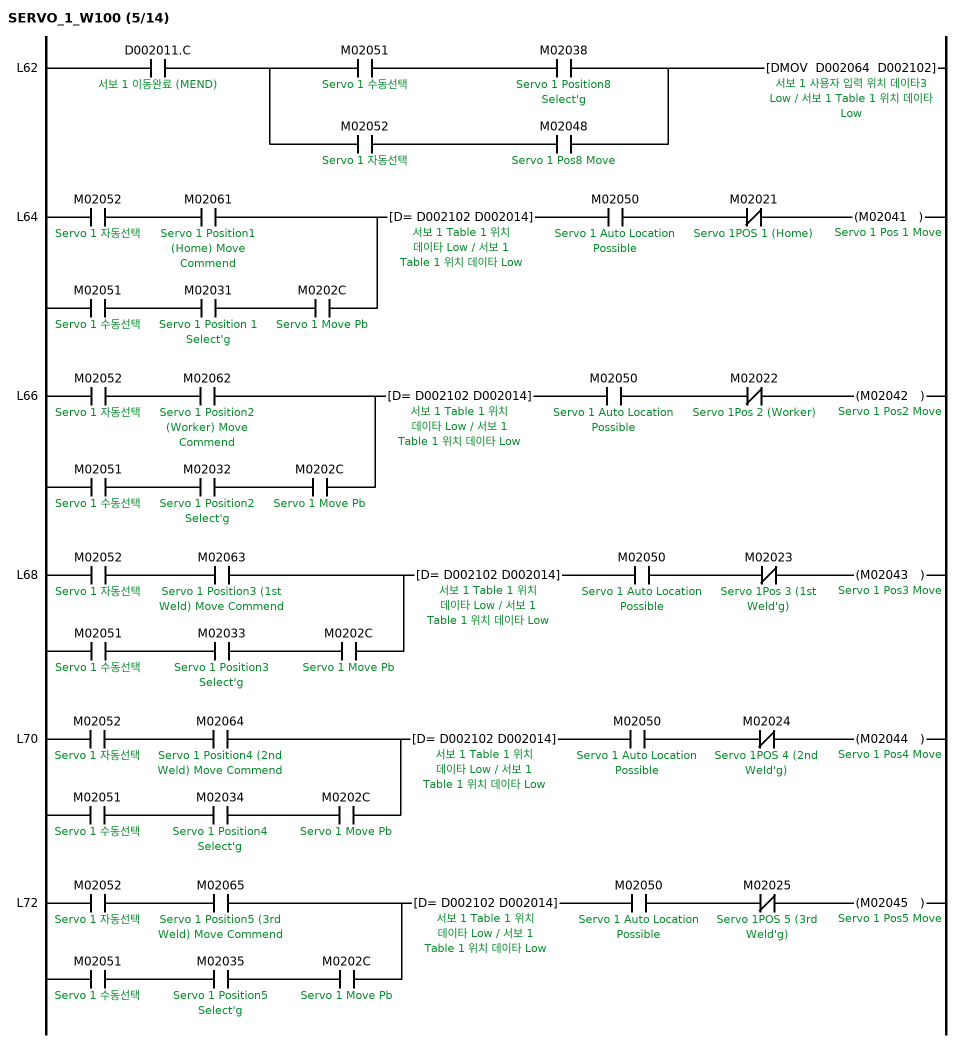
; L62
LOAD      D002011.C	// 서보 1 이동완료 (MEND)
LOAD      M02051	// Servo 1 수동선택
AND       M02038	// Servo 1 Position8 Select'g
LOAD      M02052	// Servo 1 자동선택
AND       M02048	// Servo 1 Pos8 Move
OR LOAD
AND LOAD
DMOV      D002064 D002102	// 서보 1 사용자 입력 위치 데이타3 Low / 서보 1 Table 1 위치 데이타 Low
; L64
LOAD      M02052	// Servo 1 자동선택
AND       M02061	// Servo 1 Position1 (Home) Move Commend
LOAD      M02051	// Servo 1 수동선택
AND       M02031	// Servo 1 Position 1 Select'g
AND       M0202C	// Servo 1 Move Pb
OR LOAD
ANDD=     D002102 D002014	// 서보 1 Table 1 위치 데이타 Low / 서보 1 Table 1 위치 데이타 Low
AND       M02050	// Servo 1 Auto Location Possible
AND NOT   M02021	// Servo 1POS 1 (Home)
OUT       M02041	// Servo 1 Pos 1 Move
; L66
LOAD      M02052	// Servo 1 자동선택
AND       M02062	// Servo 1 Position2 (Worker) Move Commend
LOAD      M02051	// Servo 1 수동선택
AND       M02032	// Servo 1 Position2 Select'g
AND       M0202C	// Servo 1 Move Pb
OR LOAD
ANDD=     D002102 D002014	// 서보 1 Table 1 위치 데이타 Low / 서보 1 Table 1 위치 데이타 Low
AND       M02050	// Servo 1 Auto Location Possible
AND NOT   M02022	// Servo 1Pos 2 (Worker)
OUT       M02042	// Servo 1 Pos2 Move
; L68
LOAD      M02052	// Servo 1 자동선택
AND       M02063	// Servo 1 Position3 (1st Weld) Move Commend
LOAD      M02051	// Servo 1 수동선택
AND       M02033	// Servo 1 Position3 Select'g
AND       M0202C	// Servo 1 Move Pb
OR LOAD
ANDD=     D002102 D002014	// 서보 1 Table 1 위치 데이타 Low / 서보 1 Table 1 위치 데이타 Low
AND       M02050	// Servo 1 Auto Location Possible
AND NOT   M02023	// Servo 1Pos 3 (1st Weld'g)
OUT       M02043	// Servo 1 Pos3 Move
; L70
LOAD      M02052	// Servo 1 자동선택
AND       M02064	// Servo 1 Position4 (2nd Weld) Move Commend
LOAD      M02051	// Servo 1 수동선택
AND       M02034	// Servo 1 Position4 Select'g
AND       M0202C	// Servo 1 Move Pb
OR LOAD
ANDD=     D002102 D002014	// 서보 1 Table 1 위치 데이타 Low / 서보 1 Table 1 위치 데이타 Low
AND       M02050	// Servo 1 Auto Location Possible
AND NOT   M02024	// Servo 1POS 4 (2nd Weld'g)
OUT       M02044	// Servo 1 Pos4 Move
; L72
LOAD      M02052	// Servo 1 자동선택
AND       M02065	// Servo 1 Position5 (3rd Weld) Move Commend
LOAD      M02051	// Servo 1 수동선택
AND       M02035	// Servo 1 Position5 Select'g
AND       M0202C	// Servo 1 Move Pb
OR LOAD
ANDD=     D002102 D002014	// 서보 1 Table 1 위치 데이타 Low / 서보 1 Table 1 위치 데이타 Low
AND       M02050	// Servo 1 Auto Location Possible
AND NOT   M02025	// Servo 1POS 5 (3rd Weld'g)
OUT       M02045	// Servo 1 Pos5 Move

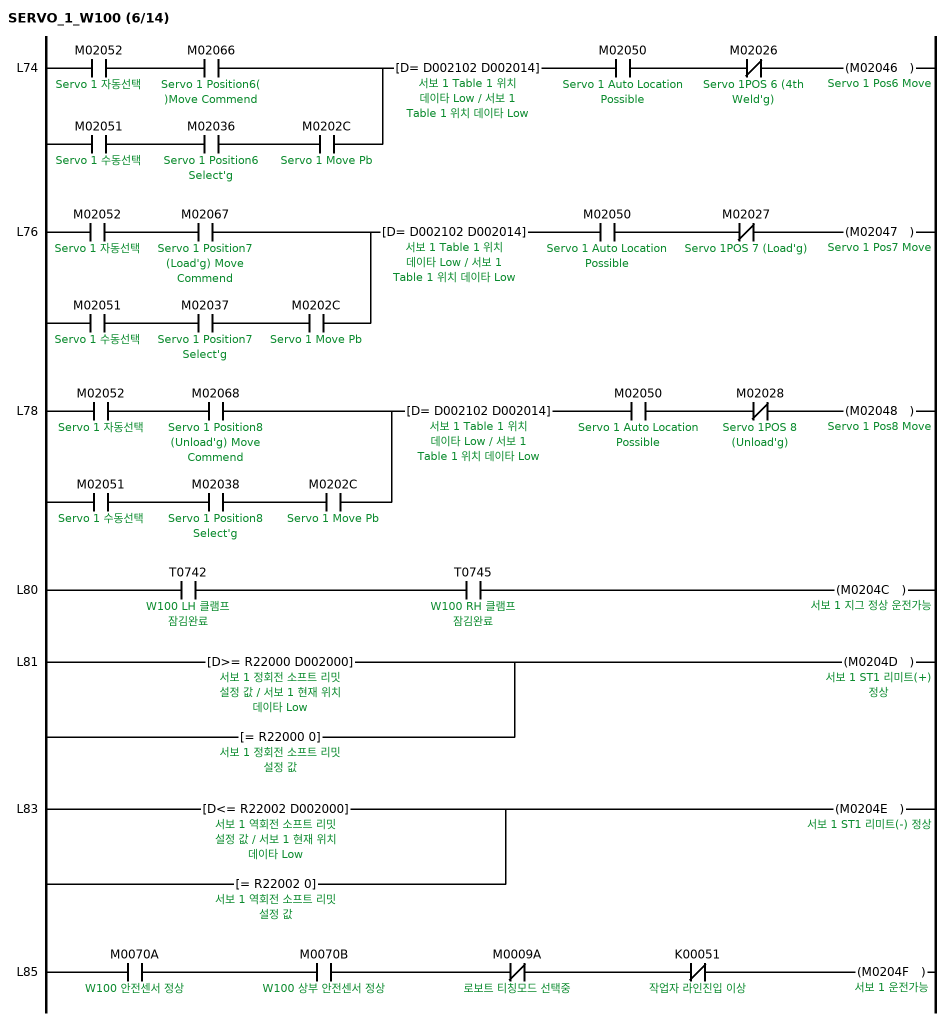
; L74
LOAD      M02052	// Servo 1 자동선택
AND       M02066	// Servo 1 Position6()Move Commend
LOAD      M02051	// Servo 1 수동선택
AND       M02036	// Servo 1 Position6 Select'g
AND       M0202C	// Servo 1 Move Pb
OR LOAD
ANDD=     D002102 D002014	// 서보 1 Table 1 위치 데이타 Low / 서보 1 Table 1 위치 데이타 Low
AND       M02050	// Servo 1 Auto Location Possible
AND NOT   M02026	// Servo 1POS 6 (4th Weld'g)
OUT       M02046	// Servo 1 Pos6 Move
; L76
LOAD      M02052	// Servo 1 자동선택
AND       M02067	// Servo 1 Position7 (Load'g) Move Commend
LOAD      M02051	// Servo 1 수동선택
AND       M02037	// Servo 1 Position7 Select'g
AND       M0202C	// Servo 1 Move Pb
OR LOAD
ANDD=     D002102 D002014	// 서보 1 Table 1 위치 데이타 Low / 서보 1 Table 1 위치 데이타 Low
AND       M02050	// Servo 1 Auto Location Possible
AND NOT   M02027	// Servo 1POS 7 (Load'g)
OUT       M02047	// Servo 1 Pos7 Move
; L78
LOAD      M02052	// Servo 1 자동선택
AND       M02068	// Servo 1 Position8 (Unload'g) Move Commend
LOAD      M02051	// Servo 1 수동선택
AND       M02038	// Servo 1 Position8 Select'g
AND       M0202C	// Servo 1 Move Pb
OR LOAD
ANDD=     D002102 D002014	// 서보 1 Table 1 위치 데이타 Low / 서보 1 Table 1 위치 데이타 Low
AND       M02050	// Servo 1 Auto Location Possible
AND NOT   M02028	// Servo 1POS 8 (Unload'g)
OUT       M02048	// Servo 1 Pos8 Move
; L80
LOAD      T0742	// W100 LH 클램프 잠김완료
AND       T0745	// W100 RH 클램프 잠김완료
OUT       M0204C	// 서보 1 지그 정상 운전가능
; L81
LOADD>=   R22000 D002000	// 서보 1 정회전 소프트 리밋 설정 값 / 서보 1 현재 위치 데이타 Low
OR=       R22000 0	// 서보 1 정회전 소프트 리밋 설정 값
OUT       M0204D	// 서보 1 ST1 리미트(+) 정상
; L83
LOADD<=   R22002 D002000	// 서보 1 역회전 소프트 리밋 설정 값 / 서보 1 현재 위치 데이타 Low
OR=       R22002 0	// 서보 1 역회전 소프트 리밋 설정 값
OUT       M0204E	// 서보 1 ST1 리미트(-) 정상
; L85
LOAD      M0070A	// W100 안전센서 정상
AND       M0070B	// W100 상부 안전센서 정상
AND NOT   M0009A	// 로보트 티칭모드 선택중
AND NOT   K00051	//  작업자 라인진입 이상
OUT       M0204F	// 서보 1 운전가능

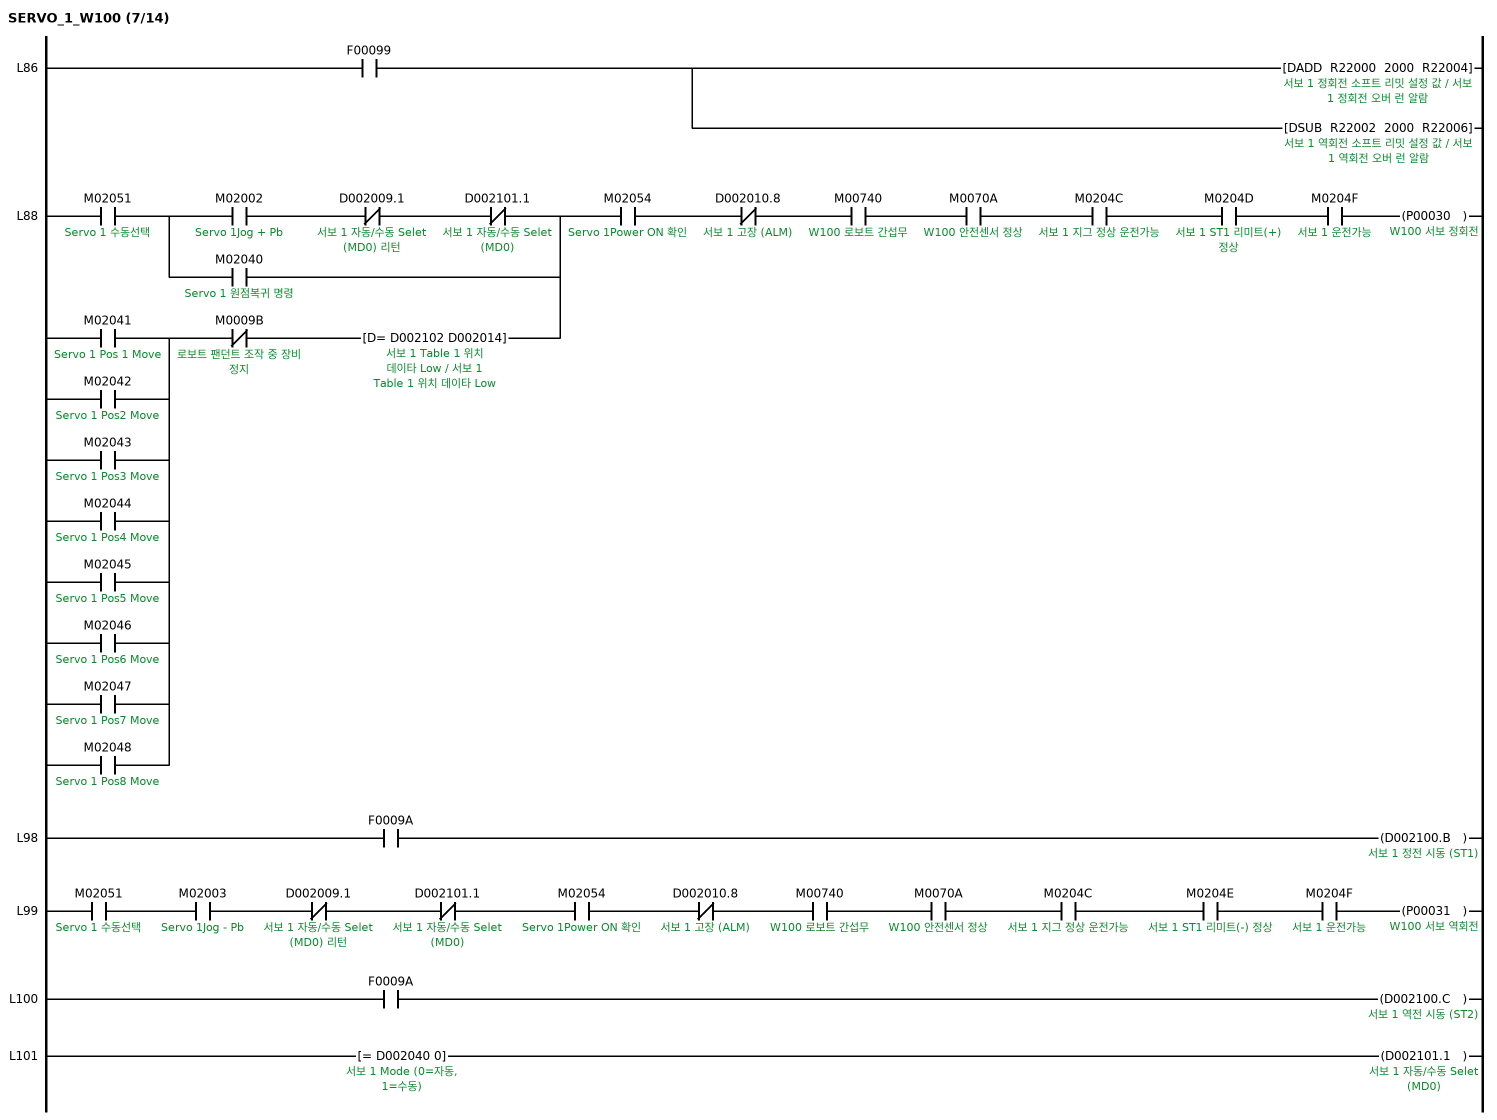
; L86
LOAD      F00099
DADD      R22000 2000 R22004	// 서보 1 정회전 소프트 리밋 설정 값 / 서보 1 정회전 오버 런 알람
DSUB      R22002 2000 R22006	// 서보 1 역회전 소프트 리밋 설정 값 / 서보 1 역회전 오버 런 알람
; L88
LOAD      M02051	// Servo 1 수동선택
LOAD      M02002	// Servo 1Jog + Pb
AND NOT   D002009.1	// 서보 1 자동/수동 Selet (MD0) 리턴
AND NOT   D002101.1	// 서보 1 자동/수동 Selet (MD0)
OR        M02040	// Servo 1 원점복귀 명령
AND LOAD
LOAD      M02041	// Servo 1 Pos 1 Move
OR        M02042	// Servo 1 Pos2 Move
OR        M02043	// Servo 1 Pos3 Move
OR        M02044	// Servo 1 Pos4 Move
OR        M02045	// Servo 1 Pos5 Move
OR        M02046	// Servo 1 Pos6 Move
OR        M02047	// Servo 1 Pos7 Move
OR        M02048	// Servo 1 Pos8 Move
AND NOT   M0009B	// 로보트 팬던트 조작 중 장비 정지
ANDD=     D002102 D002014	// 서보 1 Table 1 위치 데이타 Low / 서보 1 Table 1 위치 데이타 Low
OR LOAD
AND       M02054	// Servo 1Power ON 확인
AND NOT   D002010.8	// 서보 1 고장 (ALM)
AND       M00740	// W100 로보트 간섭무
AND       M0070A	// W100 안전센서 정상
AND       M0204C	// 서보 1 지그 정상 운전가능
AND       M0204D	// 서보 1 ST1 리미트(+) 정상
AND       M0204F	// 서보 1 운전가능
OUT       P00030	// W100 서보 정회전
; L98
LOAD      F0009A
OUT       D002100.B	// 서보 1 정전 시동 (ST1)
; L99
LOAD      M02051	// Servo 1 수동선택
AND       M02003	// Servo 1Jog - Pb
AND NOT   D002009.1	// 서보 1 자동/수동 Selet (MD0) 리턴
AND NOT   D002101.1	// 서보 1 자동/수동 Selet (MD0)
AND       M02054	// Servo 1Power ON 확인
AND NOT   D002010.8	// 서보 1 고장 (ALM)
AND       M00740	// W100 로보트 간섭무
AND       M0070A	// W100 안전센서 정상
AND       M0204C	// 서보 1 지그 정상 운전가능
AND       M0204E	// 서보 1 ST1 리미트(-) 정상
AND       M0204F	// 서보 1 운전가능
OUT       P00031	// W100 서보 역회전
; L100
LOAD      F0009A
OUT       D002100.C	// 서보 1 역전 시동 (ST2)
; L101
LOAD=     D002040 0	// 서보 1 Mode (0=자동, 1=수동)
OUT       D002101.1	// 서보 1 자동/수동 Selet (MD0)

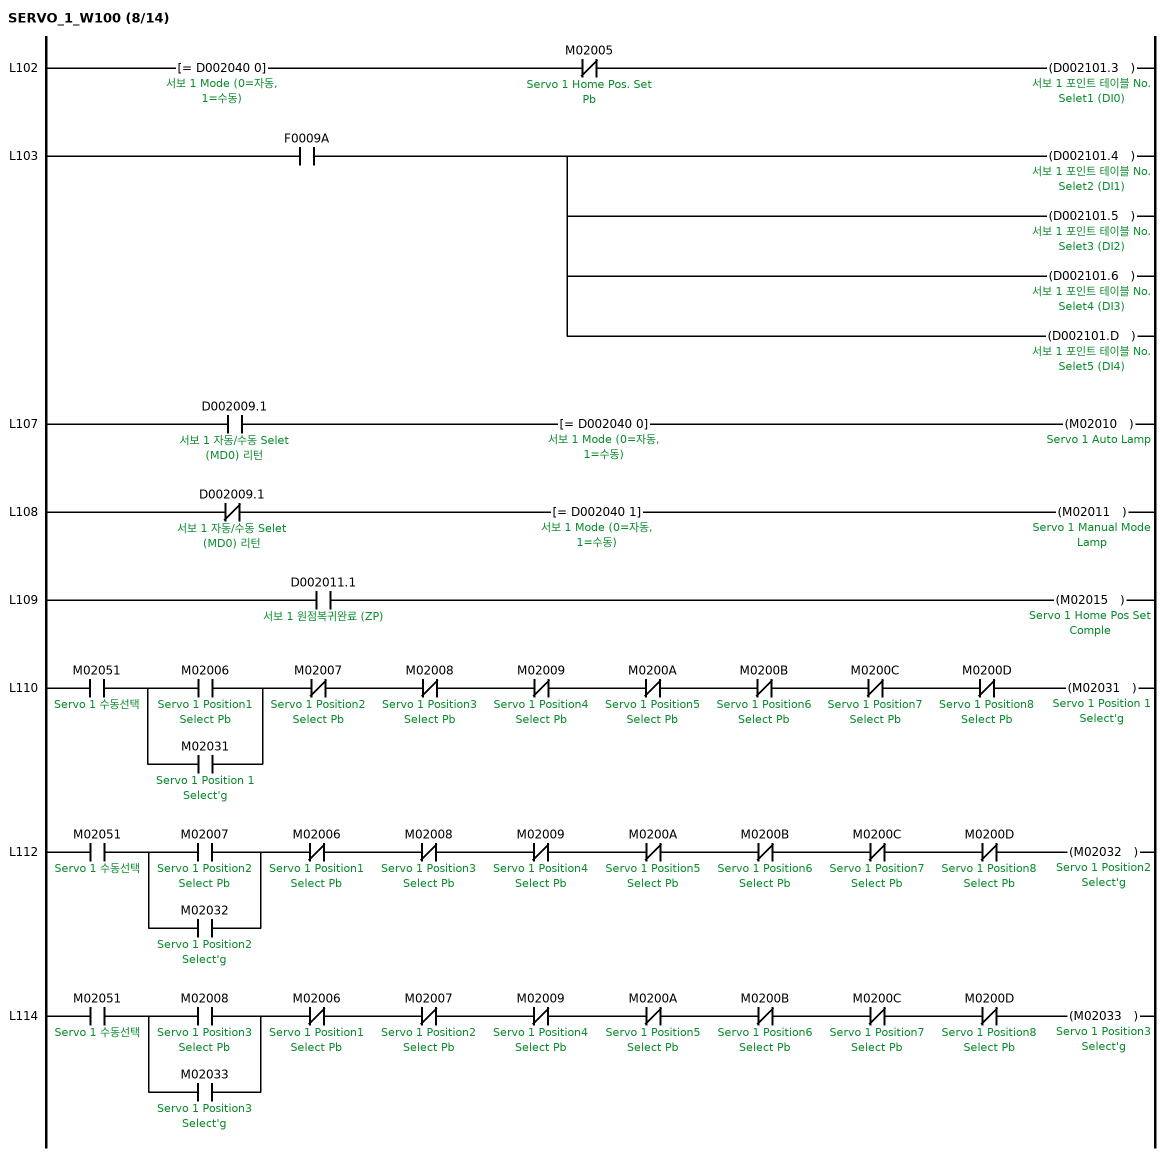
; L102
LOAD=     D002040 0	// 서보 1 Mode (0=자동, 1=수동)
AND NOT   M02005	// Servo 1 Home Pos. Set Pb
OUT       D002101.3	// 서보 1 포인트 테이블 No. Selet1 (DI0)
; L103
LOAD      F0009A
OUT       D002101.4	// 서보 1 포인트 테이블 No. Selet2 (DI1)
OUT       D002101.5	// 서보 1 포인트 테이블 No. Selet3 (DI2)
OUT       D002101.6	// 서보 1 포인트 테이블 No. Selet4 (DI3)
OUT       D002101.D	// 서보 1 포인트 테이블 No. Selet5 (DI4)
; L107
LOAD      D002009.1	// 서보 1 자동/수동 Selet (MD0) 리턴
AND=      D002040 0	// 서보 1 Mode (0=자동, 1=수동)
OUT       M02010	// Servo 1 Auto Lamp
; L108
LOAD NOT  D002009.1	// 서보 1 자동/수동 Selet (MD0) 리턴
AND=      D002040 1	// 서보 1 Mode (0=자동, 1=수동)
OUT       M02011	// Servo 1 Manual Mode Lamp
; L109
LOAD      D002011.1	// 서보 1 원점복귀완료 (ZP)
OUT       M02015	// Servo 1 Home Pos Set Comple
; L110
LOAD      M02051	// Servo 1 수동선택
LOAD      M02006	// Servo 1 Position1 Select Pb
OR        M02031	// Servo 1 Position 1 Select'g
AND LOAD
AND NOT   M02007	// Servo 1 Position2 Select Pb
AND NOT   M02008	// Servo 1 Position3 Select Pb
AND NOT   M02009	// Servo 1 Position4 Select Pb
AND NOT   M0200A	// Servo 1 Position5 Select Pb
AND NOT   M0200B	// Servo 1 Position6 Select Pb
AND NOT   M0200C	// Servo 1 Position7 Select Pb
AND NOT   M0200D	// Servo 1 Position8 Select Pb
OUT       M02031	// Servo 1 Position 1 Select'g
; L112
LOAD      M02051	// Servo 1 수동선택
LOAD      M02007	// Servo 1 Position2 Select Pb
OR        M02032	// Servo 1 Position2 Select'g
AND LOAD
AND NOT   M02006	// Servo 1 Position1 Select Pb
AND NOT   M02008	// Servo 1 Position3 Select Pb
AND NOT   M02009	// Servo 1 Position4 Select Pb
AND NOT   M0200A	// Servo 1 Position5 Select Pb
AND NOT   M0200B	// Servo 1 Position6 Select Pb
AND NOT   M0200C	// Servo 1 Position7 Select Pb
AND NOT   M0200D	// Servo 1 Position8 Select Pb
OUT       M02032	// Servo 1 Position2 Select'g
; L114
LOAD      M02051	// Servo 1 수동선택
LOAD      M02008	// Servo 1 Position3 Select Pb
OR        M02033	// Servo 1 Position3 Select'g
AND LOAD
AND NOT   M02006	// Servo 1 Position1 Select Pb
AND NOT   M02007	// Servo 1 Position2 Select Pb
AND NOT   M02009	// Servo 1 Position4 Select Pb
AND NOT   M0200A	// Servo 1 Position5 Select Pb
AND NOT   M0200B	// Servo 1 Position6 Select Pb
AND NOT   M0200C	// Servo 1 Position7 Select Pb
AND NOT   M0200D	// Servo 1 Position8 Select Pb
OUT       M02033	// Servo 1 Position3 Select'g

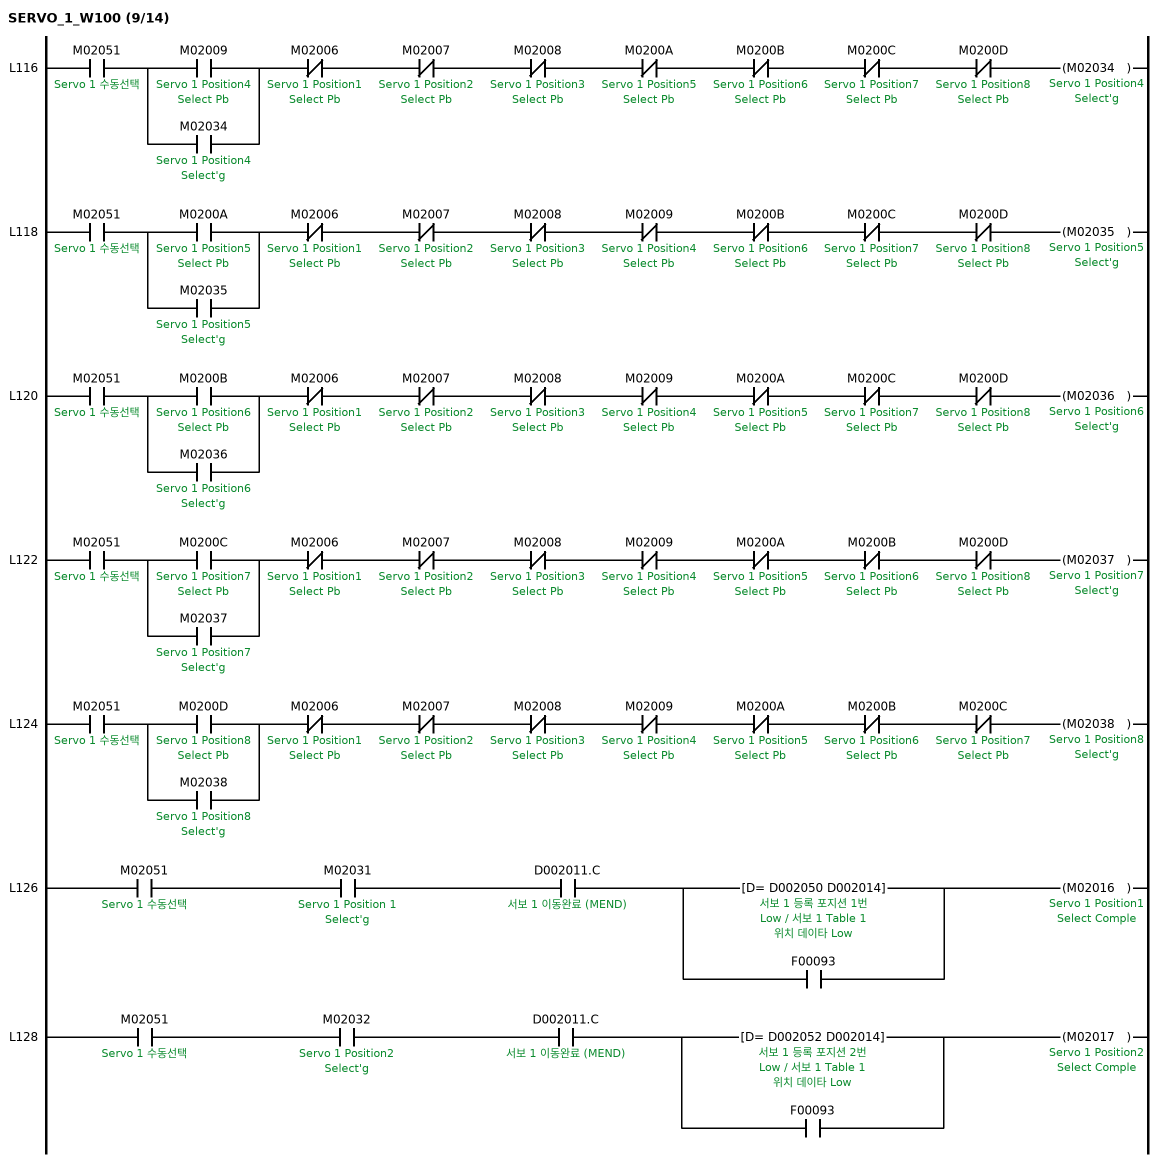
; L116
LOAD      M02051	// Servo 1 수동선택
LOAD      M02009	// Servo 1 Position4 Select Pb
OR        M02034	// Servo 1 Position4 Select'g
AND LOAD
AND NOT   M02006	// Servo 1 Position1 Select Pb
AND NOT   M02007	// Servo 1 Position2 Select Pb
AND NOT   M02008	// Servo 1 Position3 Select Pb
AND NOT   M0200A	// Servo 1 Position5 Select Pb
AND NOT   M0200B	// Servo 1 Position6 Select Pb
AND NOT   M0200C	// Servo 1 Position7 Select Pb
AND NOT   M0200D	// Servo 1 Position8 Select Pb
OUT       M02034	// Servo 1 Position4 Select'g
; L118
LOAD      M02051	// Servo 1 수동선택
LOAD      M0200A	// Servo 1 Position5 Select Pb
OR        M02035	// Servo 1 Position5 Select'g
AND LOAD
AND NOT   M02006	// Servo 1 Position1 Select Pb
AND NOT   M02007	// Servo 1 Position2 Select Pb
AND NOT   M02008	// Servo 1 Position3 Select Pb
AND NOT   M02009	// Servo 1 Position4 Select Pb
AND NOT   M0200B	// Servo 1 Position6 Select Pb
AND NOT   M0200C	// Servo 1 Position7 Select Pb
AND NOT   M0200D	// Servo 1 Position8 Select Pb
OUT       M02035	// Servo 1 Position5 Select'g
; L120
LOAD      M02051	// Servo 1 수동선택
LOAD      M0200B	// Servo 1 Position6 Select Pb
OR        M02036	// Servo 1 Position6 Select'g
AND LOAD
AND NOT   M02006	// Servo 1 Position1 Select Pb
AND NOT   M02007	// Servo 1 Position2 Select Pb
AND NOT   M02008	// Servo 1 Position3 Select Pb
AND NOT   M02009	// Servo 1 Position4 Select Pb
AND NOT   M0200A	// Servo 1 Position5 Select Pb
AND NOT   M0200C	// Servo 1 Position7 Select Pb
AND NOT   M0200D	// Servo 1 Position8 Select Pb
OUT       M02036	// Servo 1 Position6 Select'g
; L122
LOAD      M02051	// Servo 1 수동선택
LOAD      M0200C	// Servo 1 Position7 Select Pb
OR        M02037	// Servo 1 Position7 Select'g
AND LOAD
AND NOT   M02006	// Servo 1 Position1 Select Pb
AND NOT   M02007	// Servo 1 Position2 Select Pb
AND NOT   M02008	// Servo 1 Position3 Select Pb
AND NOT   M02009	// Servo 1 Position4 Select Pb
AND NOT   M0200A	// Servo 1 Position5 Select Pb
AND NOT   M0200B	// Servo 1 Position6 Select Pb
AND NOT   M0200D	// Servo 1 Position8 Select Pb
OUT       M02037	// Servo 1 Position7 Select'g
; L124
LOAD      M02051	// Servo 1 수동선택
LOAD      M0200D	// Servo 1 Position8 Select Pb
OR        M02038	// Servo 1 Position8 Select'g
AND LOAD
AND NOT   M02006	// Servo 1 Position1 Select Pb
AND NOT   M02007	// Servo 1 Position2 Select Pb
AND NOT   M02008	// Servo 1 Position3 Select Pb
AND NOT   M02009	// Servo 1 Position4 Select Pb
AND NOT   M0200A	// Servo 1 Position5 Select Pb
AND NOT   M0200B	// Servo 1 Position6 Select Pb
AND NOT   M0200C	// Servo 1 Position7 Select Pb
OUT       M02038	// Servo 1 Position8 Select'g
; L126
LOAD      M02051	// Servo 1 수동선택
AND       M02031	// Servo 1 Position 1 Select'g
AND       D002011.C	// 서보 1 이동완료 (MEND)
LOADD=    D002050 D002014	// 서보 1 등록 포지션 1번 Low / 서보 1 Table 1 위치 데이타 Low
OR        F00093
AND LOAD
OUT       M02016	// Servo 1 Position1 Select Comple
; L128
LOAD      M02051	// Servo 1 수동선택
AND       M02032	// Servo 1 Position2 Select'g
AND       D002011.C	// 서보 1 이동완료 (MEND)
LOADD=    D002052 D002014	// 서보 1 등록 포지션 2번 Low / 서보 1 Table 1 위치 데이타 Low
OR        F00093
AND LOAD
OUT       M02017	// Servo 1 Position2 Select Comple

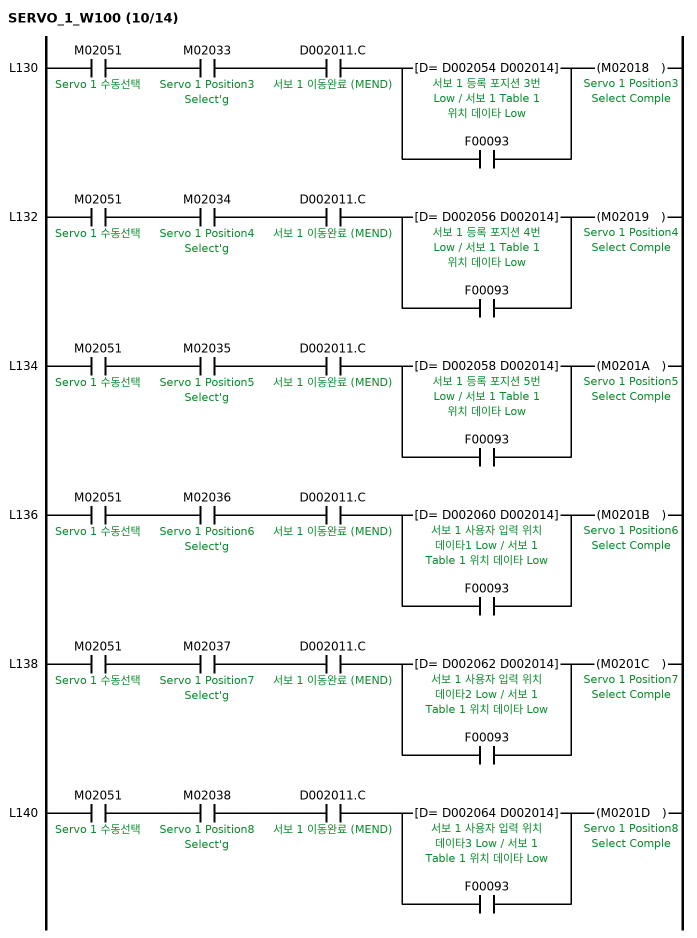
; L130
LOAD      M02051	// Servo 1 수동선택
AND       M02033	// Servo 1 Position3 Select'g
AND       D002011.C	// 서보 1 이동완료 (MEND)
LOADD=    D002054 D002014	// 서보 1 등록 포지션 3번 Low / 서보 1 Table 1 위치 데이타 Low
OR        F00093
AND LOAD
OUT       M02018	// Servo 1 Position3 Select Comple
; L132
LOAD      M02051	// Servo 1 수동선택
AND       M02034	// Servo 1 Position4 Select'g
AND       D002011.C	// 서보 1 이동완료 (MEND)
LOADD=    D002056 D002014	// 서보 1 등록 포지션 4번 Low / 서보 1 Table 1 위치 데이타 Low
OR        F00093
AND LOAD
OUT       M02019	// Servo 1 Position4 Select Comple
; L134
LOAD      M02051	// Servo 1 수동선택
AND       M02035	// Servo 1 Position5 Select'g
AND       D002011.C	// 서보 1 이동완료 (MEND)
LOADD=    D002058 D002014	// 서보 1 등록 포지션 5번 Low / 서보 1 Table 1 위치 데이타 Low
OR        F00093
AND LOAD
OUT       M0201A	// Servo 1 Position5 Select Comple
; L136
LOAD      M02051	// Servo 1 수동선택
AND       M02036	// Servo 1 Position6 Select'g
AND       D002011.C	// 서보 1 이동완료 (MEND)
LOADD=    D002060 D002014	// 서보 1 사용자 입력 위치 데이타1 Low / 서보 1 Table 1 위치 데이타 Low
OR        F00093
AND LOAD
OUT       M0201B	// Servo 1 Position6 Select Comple
; L138
LOAD      M02051	// Servo 1 수동선택
AND       M02037	// Servo 1 Position7 Select'g
AND       D002011.C	// 서보 1 이동완료 (MEND)
LOADD=    D002062 D002014	// 서보 1 사용자 입력 위치 데이타2 Low / 서보 1 Table 1 위치 데이타 Low
OR        F00093
AND LOAD
OUT       M0201C	// Servo 1 Position7 Select Comple
; L140
LOAD      M02051	// Servo 1 수동선택
AND       M02038	// Servo 1 Position8 Select'g
AND       D002011.C	// 서보 1 이동완료 (MEND)
LOADD=    D002064 D002014	// 서보 1 사용자 입력 위치 데이타3 Low / 서보 1 Table 1 위치 데이타 Low
OR        F00093
AND LOAD
OUT       M0201D	// Servo 1 Position8 Select Comple

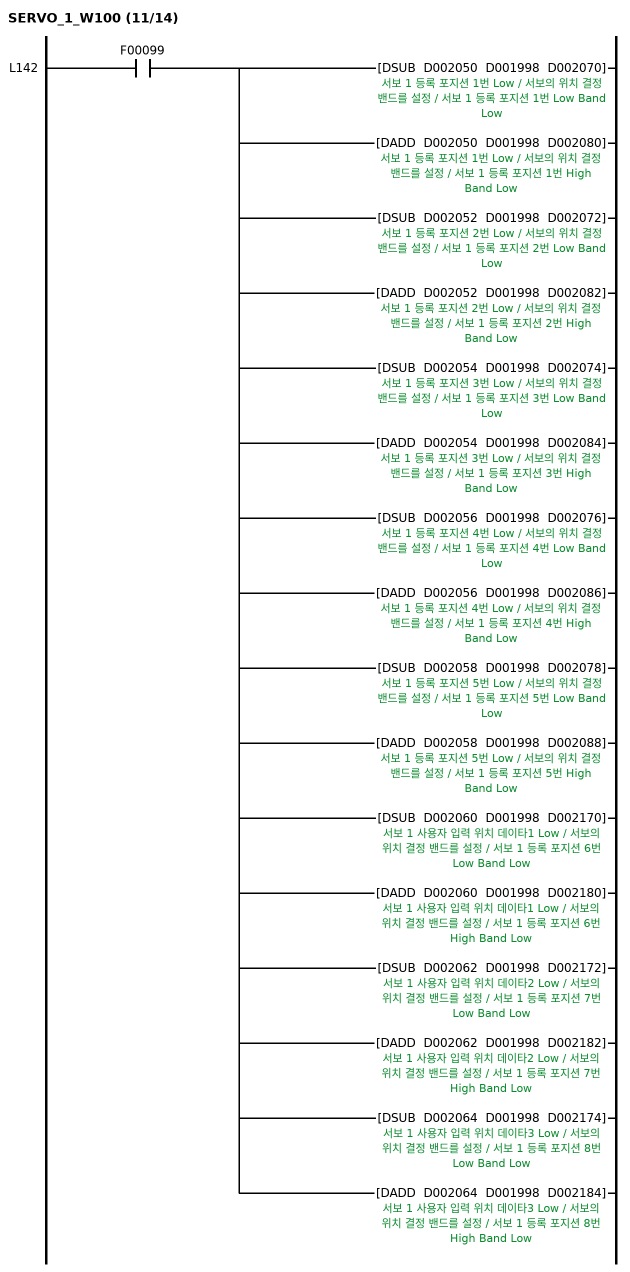
; L142
LOAD      F00099
DSUB      D002050 D001998 D002070	// 서보 1 등록 포지션 1번 Low / 서보의 위치 결정 밴드를 설정 / 서보 1 등록 포지션 1번 Low Band Low
DADD      D002050 D001998 D002080	// 서보 1 등록 포지션 1번 Low / 서보의 위치 결정 밴드를 설정 / 서보 1 등록 포지션 1번 High Band Low
DSUB      D002052 D001998 D002072	// 서보 1 등록 포지션 2번 Low / 서보의 위치 결정 밴드를 설정 / 서보 1 등록 포지션 2번 Low Band Low
DADD      D002052 D001998 D002082	// 서보 1 등록 포지션 2번 Low / 서보의 위치 결정 밴드를 설정 / 서보 1 등록 포지션 2번 High Band Low
DSUB      D002054 D001998 D002074	// 서보 1 등록 포지션 3번 Low / 서보의 위치 결정 밴드를 설정 / 서보 1 등록 포지션 3번 Low Band Low
DADD      D002054 D001998 D002084	// 서보 1 등록 포지션 3번 Low / 서보의 위치 결정 밴드를 설정 / 서보 1 등록 포지션 3번 High Band Low
DSUB      D002056 D001998 D002076	// 서보 1 등록 포지션 4번 Low / 서보의 위치 결정 밴드를 설정 / 서보 1 등록 포지션 4번 Low Band Low
DADD      D002056 D001998 D002086	// 서보 1 등록 포지션 4번 Low / 서보의 위치 결정 밴드를 설정 / 서보 1 등록 포지션 4번 High Band Low
DSUB      D002058 D001998 D002078	// 서보 1 등록 포지션 5번 Low / 서보의 위치 결정 밴드를 설정 / 서보 1 등록 포지션 5번 Low Band Low
DADD      D002058 D001998 D002088	// 서보 1 등록 포지션 5번 Low / 서보의 위치 결정 밴드를 설정 / 서보 1 등록 포지션 5번 High Band Low
DSUB      D002060 D001998 D002170	// 서보 1 사용자 입력 위치 데이타1 Low / 서보의 위치 결정 밴드를 설정 / 서보 1 등록 포지션 6번 Low Band Low
DADD      D002060 D001998 D002180	// 서보 1 사용자 입력 위치 데이타1 Low / 서보의 위치 결정 밴드를 설정 / 서보 1 등록 포지션 6번 High Band Low
DSUB      D002062 D001998 D002172	// 서보 1 사용자 입력 위치 데이타2 Low / 서보의 위치 결정 밴드를 설정 / 서보 1 등록 포지션 7번 Low Band Low
DADD      D002062 D001998 D002182	// 서보 1 사용자 입력 위치 데이타2 Low / 서보의 위치 결정 밴드를 설정 / 서보 1 등록 포지션 7번 High Band Low
DSUB      D002064 D001998 D002174	// 서보 1 사용자 입력 위치 데이타3 Low / 서보의 위치 결정 밴드를 설정 / 서보 1 등록 포지션 8번 Low Band Low
DADD      D002064 D001998 D002184	// 서보 1 사용자 입력 위치 데이타3 Low / 서보의 위치 결정 밴드를 설정 / 서보 1 등록 포지션 8번 High Band Low

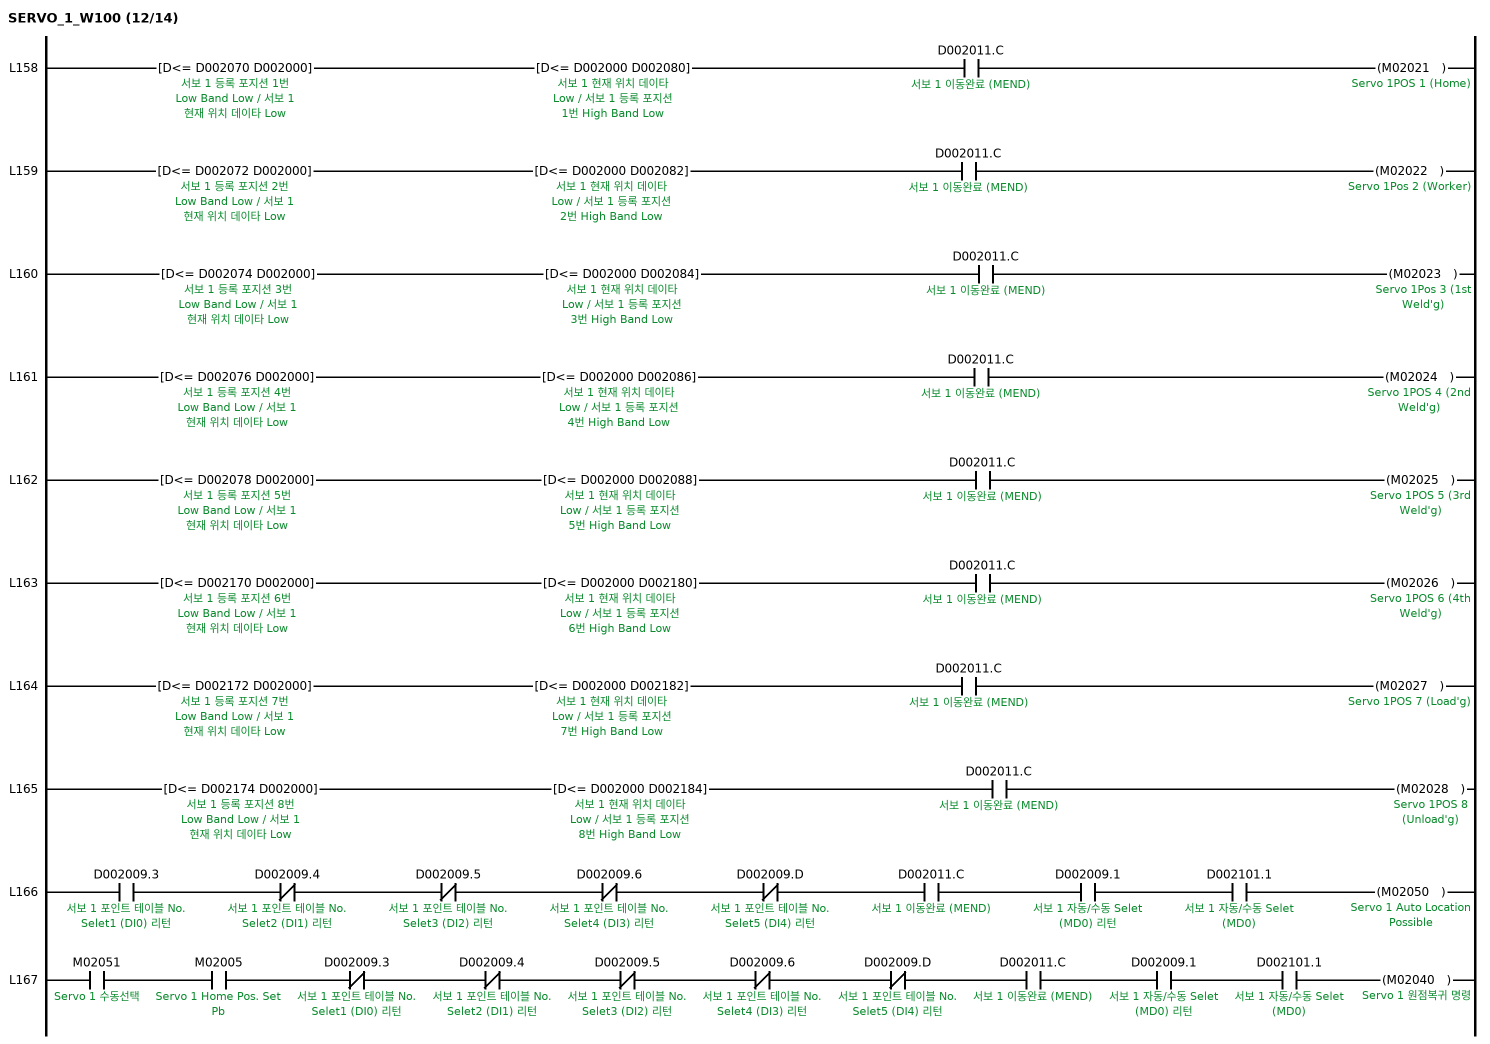
; L158
LOADD<=   D002070 D002000	// 서보 1 등록 포지션 1번 Low Band Low / 서보 1 현재 위치 데이타 Low
ANDD<=    D002000 D002080	// 서보 1 현재 위치 데이타 Low / 서보 1 등록 포지션 1번 High Band Low
AND       D002011.C	// 서보 1 이동완료 (MEND)
OUT       M02021	// Servo 1POS 1 (Home)
; L159
LOADD<=   D002072 D002000	// 서보 1 등록 포지션 2번 Low Band Low / 서보 1 현재 위치 데이타 Low
ANDD<=    D002000 D002082	// 서보 1 현재 위치 데이타 Low / 서보 1 등록 포지션 2번 High Band Low
AND       D002011.C	// 서보 1 이동완료 (MEND)
OUT       M02022	// Servo 1Pos 2 (Worker)
; L160
LOADD<=   D002074 D002000	// 서보 1 등록 포지션 3번 Low Band Low / 서보 1 현재 위치 데이타 Low
ANDD<=    D002000 D002084	// 서보 1 현재 위치 데이타 Low / 서보 1 등록 포지션 3번 High Band Low
AND       D002011.C	// 서보 1 이동완료 (MEND)
OUT       M02023	// Servo 1Pos 3 (1st Weld'g)
; L161
LOADD<=   D002076 D002000	// 서보 1 등록 포지션 4번 Low Band Low / 서보 1 현재 위치 데이타 Low
ANDD<=    D002000 D002086	// 서보 1 현재 위치 데이타 Low / 서보 1 등록 포지션 4번 High Band Low
AND       D002011.C	// 서보 1 이동완료 (MEND)
OUT       M02024	// Servo 1POS 4 (2nd Weld'g)
; L162
LOADD<=   D002078 D002000	// 서보 1 등록 포지션 5번 Low Band Low / 서보 1 현재 위치 데이타 Low
ANDD<=    D002000 D002088	// 서보 1 현재 위치 데이타 Low / 서보 1 등록 포지션 5번 High Band Low
AND       D002011.C	// 서보 1 이동완료 (MEND)
OUT       M02025	// Servo 1POS 5 (3rd Weld'g)
; L163
LOADD<=   D002170 D002000	// 서보 1 등록 포지션 6번 Low Band Low / 서보 1 현재 위치 데이타 Low
ANDD<=    D002000 D002180	// 서보 1 현재 위치 데이타 Low / 서보 1 등록 포지션 6번 High Band Low
AND       D002011.C	// 서보 1 이동완료 (MEND)
OUT       M02026	// Servo 1POS 6 (4th Weld'g)
; L164
LOADD<=   D002172 D002000	// 서보 1 등록 포지션 7번 Low Band Low / 서보 1 현재 위치 데이타 Low
ANDD<=    D002000 D002182	// 서보 1 현재 위치 데이타 Low / 서보 1 등록 포지션 7번 High Band Low
AND       D002011.C	// 서보 1 이동완료 (MEND)
OUT       M02027	// Servo 1POS 7 (Load'g)
; L165
LOADD<=   D002174 D002000	// 서보 1 등록 포지션 8번 Low Band Low / 서보 1 현재 위치 데이타 Low
ANDD<=    D002000 D002184	// 서보 1 현재 위치 데이타 Low / 서보 1 등록 포지션 8번 High Band Low
AND       D002011.C	// 서보 1 이동완료 (MEND)
OUT       M02028	// Servo 1POS 8 (Unload'g)
; L166
LOAD      D002009.3	// 서보 1 포인트 테이블 No. Selet1 (DI0) 리턴
AND NOT   D002009.4	// 서보 1 포인트 테이블 No. Selet2 (DI1) 리턴
AND NOT   D002009.5	// 서보 1 포인트 테이블 No. Selet3 (DI2) 리턴
AND NOT   D002009.6	// 서보 1 포인트 테이블 No. Selet4 (DI3) 리턴
AND NOT   D002009.D	// 서보 1 포인트 테이블 No. Selet5 (DI4) 리턴
AND       D002011.C	// 서보 1 이동완료 (MEND)
AND       D002009.1	// 서보 1 자동/수동 Selet (MD0) 리턴
AND       D002101.1	// 서보 1 자동/수동 Selet (MD0)
OUT       M02050	// Servo 1 Auto Location Possible
; L167
LOAD      M02051	// Servo 1 수동선택
AND       M02005	// Servo 1 Home Pos. Set Pb
AND NOT   D002009.3	// 서보 1 포인트 테이블 No. Selet1 (DI0) 리턴
AND NOT   D002009.4	// 서보 1 포인트 테이블 No. Selet2 (DI1) 리턴
AND NOT   D002009.5	// 서보 1 포인트 테이블 No. Selet3 (DI2) 리턴
AND NOT   D002009.6	// 서보 1 포인트 테이블 No. Selet4 (DI3) 리턴
AND NOT   D002009.D	// 서보 1 포인트 테이블 No. Selet5 (DI4) 리턴
AND       D002011.C	// 서보 1 이동완료 (MEND)
AND       D002009.1	// 서보 1 자동/수동 Selet (MD0) 리턴
AND       D002101.1	// 서보 1 자동/수동 Selet (MD0)
OUT       M02040	// Servo 1 원점복귀 명령

